KUKA KRL program: f1_Kuka_APT216T03S16.SRC

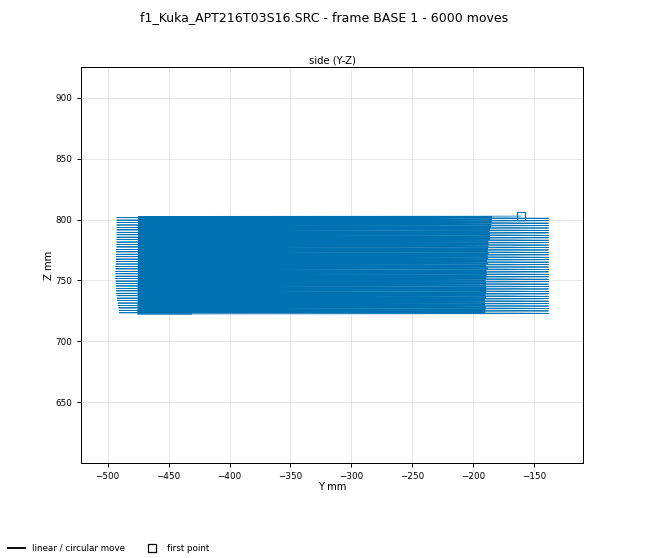
[picture p0: tool path of f1_Kuka_APT216T03S16.SRC in frame BASE 1, 6000 of 6001 moves have a stored position in this frame; points joined in program order, loops and branches not executed]
&ACCESS RVP
&REL 2
&PARAM TEMPLATE = C:\KRC\Roboter\Template\vorgabe
&PARAM EDITMASK = *
DEF f1_Kuka_APT216T03S16()


;FOLD INI;%{PE}%V3.2.0,%MKUKATPBASIS,%CINIT,%VCOMMON,%P
  ;FOLD BAS INI;%{E}%V3.2.0,%MKUKATPBASIS,%CINIT,%VINIT,%P
    GLOBAL INTERRUPT DECL 3 WHEN $STOPMESS==TRUE DO IR_STOPM ( )
    INTERRUPT ON 3
    BAS (#INITMOV,0 )
  ;ENDFOLD (BAS INI)
  ;FOLD USER INI;%{E}%V3.2.0,%MKUKATPUSER,%CINIT,%VINIT,%P
    ;Make your modifications here
  ;ENDFOLD (USER INI)
;ENDFOLD (INI)


;*** Make Null PTP Move
  PTP $pos_act

;*** Auto Load The Correct TOOL Data
  $tool=tool_data[3]

;*** Auto Load The Correct BASE Data
  $base=base_data[1]

  $ADVANCE = 5

;*** Restate Last Velocity
MMPM(30000.0)
SetRPM(6000)
LIN {X -0.024,Y -161.232,Z 802.830,A 0.000,B 0.000,C 90.000,E1 149.459} C_DIS
LIN {X 0.060,Y -163.319,Z 802.820,A 0.000,B 0.000,C 90.000,E1 147.661} C_DIS
LIN {X -0.068,Y -167.771,Z 802.801,A 0.000,B 0.000,C 90.000,E1 144.196} C_DIS
LIN {X 0.084,Y -171.586,Z 802.786,A 0.000,B 0.000,C 90.000,E1 141.537} C_DIS
LIN {X 0.015,Y -176.537,Z 802.767,A 0.000,B 0.000,C 90.000,E1 138.119} C_DIS
LIN {X 0.007,Y -180.836,Z 802.753,A 0.000,B 0.000,C 90.000,E1 135.567} C_DIS
LIN {X -0.008,Y -186.246,Z 802.734,A 0.000,B 0.000,C 90.000,E1 132.204} C_DIS
LIN {X -0.071,Y -190.882,Z 802.721,A 0.000,B 0.000,C 90.000,E1 129.725} C_DIS
LIN {X 0.062,Y -192.636,Z 802.715,A 0.000,B 0.000,C 90.000,E1 128.624} C_DIS
LIN {X 0.046,Y -293.294,Z 802.715,A 0.000,B 0.000,C 90.000,E1 128.624} C_DIS
LIN {X -0.102,Y -294.709,Z 802.714,A 0.000,B 0.000,C 90.000,E1 128.624} C_DIS
LIN {X -0.048,Y -299.870,Z 802.713,A 0.000,B 0.000,C 90.000,E1 128.338} C_DIS
LIN {X 0.009,Y -302.645,Z 802.711,A 0.000,B 0.000,C 90.000,E1 128.051} C_DIS
LIN {X -0.181,Y -306.338,Z 802.708,A 0.000,B 0.000,C 90.000,E1 127.523} C_DIS
LIN {X 0.019,Y -307.841,Z 802.706,A 0.000,B 0.000,C 90.000,E1 127.156} C_DIS
LIN {X 0.036,Y -309.022,Z 802.705,A 0.000,B 0.000,C 90.000,E1 126.824} C_DIS
LIN {X -0.142,Y -320.038,Z 802.685,A 0.000,B 0.000,C 90.000,E1 123.293} C_DIS
LIN {X -0.035,Y -330.415,Z 802.669,A 0.000,B 0.000,C 90.000,E1 120.413} C_DIS
LIN {X 0.057,Y -342.138,Z 802.653,A 0.000,B 0.000,C 90.000,E1 117.590} C_DIS
LIN {X 0.009,Y -355.318,Z 802.638,A 0.000,B 0.000,C 90.000,E1 114.847} C_DIS
LIN {X -0.042,Y -368.347,Z 802.625,A 0.000,B 0.000,C 90.000,E1 112.461} C_DIS
LIN {X -0.058,Y -382.712,Z 802.612,A 0.000,B 0.000,C 90.000,E1 110.120} C_DIS
LIN {X 0.023,Y -398.513,Z 802.599,A 0.000,B 0.000,C 90.000,E1 107.819} C_DIS
LIN {X -0.127,Y -415.866,Z 802.587,A 0.000,B 0.000,C 90.000,E1 105.607} C_DIS
LIN {X 0.032,Y -434.898,Z 802.575,A 0.000,B 0.000,C 90.000,E1 103.411} C_DIS
LIN {X 0.068,Y -454.991,Z 802.563,A 0.000,B 0.000,C 90.000,E1 101.366} C_DIS
LIN {X -0.083,Y -467.781,Z 802.557,A 0.000,B 0.000,C 90.000,E1 100.197} C_DIS
LIN {X -0.048,Y -469.816,Z 802.555,A 0.000,B 0.000,C 90.000,E1 99.962} C_DIS
LIN {X -0.200,Y -471.497,Z 802.554,A 0.000,B 0.000,C 90.000,E1 99.726} C_DIS
LIN {X 0.036,Y -472.760,Z 802.552,A 0.000,B 0.000,C 90.000,E1 99.443} C_DIS
LIN {X 0.218,Y -474.319,Z 802.550,A 0.000,B 0.000,C 90.000,E1 98.916} C_DIS
LIN {X -0.134,Y -474.830,Z 802.547,A 0.000,B 0.000,C 90.000,E1 98.454} C_DIS
LIN {X -0.007,Y -474.378,Z 802.544,A 0.000,B 0.000,C 90.000,E1 97.936} C_DIS
LIN {X 0.185,Y -472.896,Z 802.541,A 0.000,B 0.000,C 90.000,E1 97.409} C_DIS
LIN {X -0.015,Y -471.693,Z 802.540,A 0.000,B 0.000,C 90.000,E1 97.182} C_DIS
LIN {X 0.161,Y -454.007,Z 802.524,A 0.000,B 0.000,C 90.000,E1 94.359} C_DIS
LIN {X -0.210,Y -440.415,Z 802.511,A 0.000,B 0.000,C 90.000,E1 92.064} C_DIS
LIN {X -0.069,Y -431.096,Z 802.503,A 0.000,B 0.000,C 90.000,E1 90.458} C_DIS
LIN {X 0.016,Y -419.942,Z 802.492,A 0.000,B 0.000,C 90.000,E1 88.568} C_DIS
LIN {X -0.207,Y -410.228,Z 802.483,A 0.000,B 0.000,C 90.000,E1 86.963} C_DIS
LIN {X -0.090,Y -398.712,Z 802.472,A 0.000,B 0.000,C 90.000,E1 85.008} C_DIS
LIN {X -0.164,Y -385.665,Z 802.460,A 0.000,B 0.000,C 90.000,E1 82.761} C_DIS
LIN {X -0.060,Y -371.493,Z 802.445,A 0.000,B 0.000,C 90.000,E1 80.151} C_DIS
LIN {X 0.105,Y -356.306,Z 802.429,A 0.000,B 0.000,C 90.000,E1 77.173} C_DIS
LIN {X 0.123,Y -344.660,Z 802.415,A 0.000,B 0.000,C 90.000,E1 74.755} C_DIS
LIN {X 0.037,Y -333.108,Z 802.402,A 0.000,B 0.000,C 90.000,E1 72.308} C_DIS
LIN {X -0.175,Y -320.385,Z 802.386,A 0.000,B 0.000,C 90.000,E1 69.518} C_DIS
LIN {X -0.054,Y -306.773,Z 802.368,A 0.000,B 0.000,C 90.000,E1 66.282} C_DIS
LIN {X -0.094,Y -294.227,Z 802.350,A 0.000,B 0.000,C 90.000,E1 62.999} C_DIS
LIN {X 0.029,Y -283.577,Z 802.333,A 0.000,B 0.000,C 90.000,E1 59.950} C_DIS
LIN {X 0.171,Y -273.514,Z 802.316,A 0.000,B 0.000,C 90.000,E1 56.834} C_DIS
LIN {X 0.145,Y -265.985,Z 802.302,A 0.000,B 0.000,C 90.000,E1 54.402} C_DIS
LIN {X 0.011,Y -259.636,Z 802.291,A 0.000,B 0.000,C 90.000,E1 52.316} C_DIS
LIN {X -0.014,Y -251.225,Z 802.275,A 0.000,B 0.000,C 90.000,E1 49.461} C_DIS
LIN {X 0.018,Y -241.238,Z 802.255,A 0.000,B 0.000,C 90.000,E1 45.810} C_DIS
LIN {X 0.075,Y -232.062,Z 802.234,A 0.000,B 0.000,C 90.000,E1 42.081} C_DIS
LIN {X 0.021,Y -225.008,Z 802.217,A 0.000,B 0.000,C 90.000,E1 39.072} C_DIS
LIN {X 0.019,Y -216.511,Z 802.196,A 0.000,B 0.000,C 90.000,E1 35.231} C_DIS
LIN {X -0.068,Y -210.188,Z 802.178,A 0.000,B 0.000,C 90.000,E1 32.133} C_DIS
LIN {X 0.005,Y -204.534,Z 802.161,A 0.000,B 0.000,C 90.000,E1 28.949} C_DIS
LIN {X 0.099,Y -199.559,Z 802.143,A 0.000,B 0.000,C 90.000,E1 25.720} C_DIS
LIN {X -0.011,Y -195.325,Z 802.125,A 0.000,B 0.000,C 90.000,E1 22.514} C_DIS
LIN {X 0.021,Y -191.093,Z 802.102,A 0.000,B 0.000,C 90.000,E1 18.417} C_DIS
LIN {X -0.033,Y -187.480,Z 802.075,A 0.000,B 0.000,C 90.000,E1 13.480} C_DIS
LIN {X -0.067,Y -185.036,Z 802.038,A 0.000,B 0.000,C 90.000,E1 6.834} C_DIS
LIN {X 0.017,Y -186.593,Z 801.974,A 0.000,B 0.000,C 90.000,E1 355.355} C_DIS
LIN {X -0.039,Y -189.431,Z 801.947,A 0.000,B 0.000,C 90.000,E1 350.387} C_DIS
LIN {X 0.059,Y -193.534,Z 801.919,A 0.000,B 0.000,C 90.000,E1 345.408} C_DIS
LIN {X 0.027,Y -197.946,Z 801.896,A 0.000,B 0.000,C 90.000,E1 341.329} C_DIS
LIN {X 0.027,Y -203.325,Z 801.874,A 0.000,B 0.000,C 90.000,E1 337.283} C_DIS
LIN {X 0.047,Y -208.352,Z 801.856,A 0.000,B 0.000,C 90.000,E1 334.076} C_DIS
LIN {X -0.005,Y -214.072,Z 801.838,A 0.000,B 0.000,C 90.000,E1 330.923} C_DIS
LIN {X -0.088,Y -221.910,Z 801.817,A 0.000,B 0.000,C 90.000,E1 327.041} C_DIS
LIN {X 0.131,Y -228.708,Z 801.800,A 0.000,B 0.000,C 90.000,E1 323.909} C_DIS
LIN {X 0.035,Y -237.880,Z 801.779,A 0.000,B 0.000,C 90.000,E1 320.150} C_DIS
LIN {X -0.020,Y -246.975,Z 801.760,A 0.000,B 0.000,C 90.000,E1 316.824} C_DIS
LIN {X 0.009,Y -256.777,Z 801.742,A 0.000,B 0.000,C 90.000,E1 313.542} C_DIS
LIN {X -0.010,Y -267.270,Z 801.724,A 0.000,B 0.000,C 90.000,E1 310.334} C_DIS
LIN {X -0.144,Y -280.020,Z 801.705,A 0.000,B 0.000,C 90.000,E1 306.870} C_DIS
LIN {X -0.053,Y -291.202,Z 801.690,A 0.000,B 0.000,C 90.000,E1 304.119} C_DIS
LIN {X -0.149,Y -305.021,Z 801.673,A 0.000,B 0.000,C 90.000,E1 301.131} C_DIS
LIN {X -0.014,Y -316.931,Z 801.660,A 0.000,B 0.000,C 90.000,E1 298.821} C_DIS
LIN {X -0.144,Y -333.668,Z 801.644,A 0.000,B 0.000,C 90.000,E1 295.976} C_DIS
LIN {X 0.062,Y -349.615,Z 801.630,A 0.000,B 0.000,C 90.000,E1 293.462} C_DIS
LIN {X 0.090,Y -367.192,Z 801.617,A 0.000,B 0.000,C 90.000,E1 291.046} C_DIS
LIN {X 0.108,Y -391.664,Z 801.601,A 0.000,B 0.000,C 90.000,E1 288.127} C_DIS
LIN {X 0.031,Y -409.097,Z 801.590,A 0.000,B 0.000,C 90.000,E1 286.205} C_DIS
LIN {X 0.102,Y -421.589,Z 801.582,A 0.000,B 0.000,C 90.000,E1 284.828} C_DIS
LIN {X -0.046,Y -431.397,Z 801.576,A 0.000,B 0.000,C 90.000,E1 283.772} C_DIS
LIN {X 0.161,Y -443.375,Z 801.569,A 0.000,B 0.000,C 90.000,E1 282.411} C_DIS
LIN {X 0.111,Y -452.462,Z 801.563,A 0.000,B 0.000,C 90.000,E1 281.366} C_DIS
LIN {X -0.193,Y -460.841,Z 801.557,A 0.000,B 0.000,C 90.000,E1 280.366} C_DIS
LIN {X -0.037,Y -468.618,Z 801.552,A 0.000,B 0.000,C 90.000,E1 279.321} C_DIS
LIN {X -0.111,Y -474.039,Z 801.548,A 0.000,B 0.000,C 90.000,E1 278.568} C_DIS
LIN {X -0.134,Y -478.846,Z 801.543,A 0.000,B 0.000,C 90.000,E1 277.814} C_DIS
LIN {X -0.180,Y -482.999,Z 801.539,A 0.000,B 0.000,C 90.000,E1 277.068} C_DIS
LIN {X -0.125,Y -486.497,Z 801.535,A 0.000,B 0.000,C 90.000,E1 276.315} C_DIS
LIN {X -0.095,Y -489.290,Z 801.531,A 0.000,B 0.000,C 90.000,E1 275.568} C_DIS
LIN {X 0.114,Y -490.692,Z 801.528,A 0.000,B 0.000,C 90.000,E1 275.049} C_DIS
LIN {X -0.158,Y -491.677,Z 801.525,A 0.000,B 0.000,C 90.000,E1 274.588} C_DIS
LIN {X 0.032,Y -492.321,Z 801.523,A 0.000,B 0.000,C 90.000,E1 274.073} C_DIS
LIN {X -0.229,Y -492.497,Z 801.520,A 0.000,B 0.000,C 90.000,E1 273.612} C_DIS
LIN {X 0.001,Y -492.328,Z 801.517,A 0.000,B 0.000,C 90.000,E1 273.094} C_DIS
LIN {X 0.206,Y -491.749,Z 801.514,A 0.000,B 0.000,C 90.000,E1 272.579} C_DIS
LIN {X -0.079,Y -490.766,Z 801.512,A 0.000,B 0.000,C 90.000,E1 272.121} C_DIS
LIN {X 0.141,Y -489.390,Z 801.509,A 0.000,B 0.000,C 90.000,E1 271.604} C_DIS
LIN {X -0.150,Y -487.564,Z 801.506,A 0.000,B 0.000,C 90.000,E1 271.146} C_DIS
LIN {X 0.040,Y -485.253,Z 801.504,A 0.000,B 0.000,C 90.000,E1 270.630} C_DIS
LIN {X 0.212,Y -482.387,Z 801.501,A 0.000,B 0.000,C 90.000,E1 270.115} C_DIS
LIN {X -0.110,Y -478.964,Z 801.498,A 0.000,B 0.000,C 90.000,E1 269.656} C_DIS
LIN {X 0.029,Y -474.681,Z 801.495,A 0.000,B 0.000,C 90.000,E1 269.141} C_DIS
LIN {X 0.143,Y -469.391,Z 801.492,A 0.000,B 0.000,C 90.000,E1 268.625} C_DIS
LIN {X 0.125,Y -466.571,Z 801.491,A 0.000,B 0.000,C 90.000,E1 268.396} C_DIS
LIN {X -0.091,Y -460.311,Z 801.489,A 0.000,B 0.000,C 90.000,E1 267.993} C_DIS
LIN {X 0.156,Y -456.765,Z 801.488,A 0.000,B 0.000,C 90.000,E1 267.764} C_DIS
LIN {X -0.162,Y -449.428,Z 801.486,A 0.000,B 0.000,C 90.000,E1 267.478} C_DIS
LIN {X 0.099,Y -441.906,Z 801.484,A 0.000,B 0.000,C 90.000,E1 267.192} C_DIS
LIN {X -0.084,Y -433.510,Z 801.483,A 0.000,B 0.000,C 90.000,E1 267.020} C_DIS
LIN {X 0.009,Y -425.926,Z 801.483,A 0.000,B 0.000,C 90.000,E1 266.906} C_DIS
LIN {X 0.122,Y -418.652,Z 801.483,A 0.000,B 0.000,C 90.000,E1 266.849} C_DIS
LIN {X 0.039,Y -180.978,Z 801.483,A 0.000,B 0.000,C 90.000,E1 266.846} C_DIS
LIN {X 0.015,Y -180.886,Z 801.473,A 0.000,B 0.000,C 90.000,E1 265.122} C_DIS
LIN {X 0.074,Y -179.008,Z 801.445,A 0.000,B 0.000,C 90.000,E1 260.038} C_DIS
LIN {X -0.008,Y -178.618,Z 801.440,A 0.000,B 0.000,C 90.000,E1 259.218} C_DIS
LIN {X 0.060,Y -175.670,Z 801.412,A 0.000,B 0.000,C 90.000,E1 254.102} C_DIS
LIN {X 0.065,Y -172.386,Z 801.388,A 0.000,B 0.000,C 90.000,E1 249.826} C_DIS
LIN {X 0.079,Y -171.189,Z 801.378,A 0.000,B 0.000,C 90.000,E1 248.103} C_DIS
LIN {X -0.029,Y -167.480,Z 801.354,A 0.000,B 0.000,C 90.000,E1 243.819} C_DIS
LIN {X -0.021,Y -166.876,Z 801.350,A 0.000,B 0.000,C 90.000,E1 242.948} C_DIS
LIN {X -0.028,Y -162.181,Z 801.321,A 0.000,B 0.000,C 90.000,E1 237.709} C_DIS
LIN {X 0.029,Y -160.748,Z 801.311,A 0.000,B 0.000,C 90.000,E1 235.928} C_DIS
LIN {X 0.007,Y -157.548,Z 801.291,A 0.000,B 0.000,C 90.000,E1 232.396} C_DIS
LIN {X -0.054,Y -155.576,Z 801.276,A 0.000,B 0.000,C 90.000,E1 229.747} C_DIS
LIN {X -0.002,Y -151.861,Z 801.251,A 0.000,B 0.000,C 90.000,E1 225.243} C_DIS
LIN {X 0.012,Y -150.084,Z 801.236,A 0.000,B 0.000,C 90.000,E1 222.528} C_DIS
LIN {X 0.046,Y -146.887,Z 801.211,A 0.000,B 0.000,C 90.000,E1 217.971} C_DIS
LIN {X 0.034,Y -145.473,Z 801.196,A 0.000,B 0.000,C 90.000,E1 215.231} C_DIS
LIN {X -0.049,Y -142.884,Z 801.170,A 0.000,B 0.000,C 90.000,E1 210.669} C_DIS
LIN {X 0.008,Y -141.503,Z 801.150,A 0.000,B 0.000,C 90.000,E1 206.950} C_DIS
LIN {X 0.056,Y -139.389,Z 801.114,A 0.000,B 0.000,C 90.000,E1 200.429} C_DIS
LIN {X -0.024,Y -139.096,Z 801.103,A 0.000,B 0.000,C 90.000,E1 198.598} C_DIS
LIN {X -0.031,Y -138.354,Z 801.057,A 0.000,B 0.000,C 90.000,E1 190.197} C_DIS
LIN {X -0.039,Y -139.516,Z 801.005,A 0.000,B 0.000,C 90.000,E1 180.859} C_DIS
LIN {X 0.042,Y -141.170,Z 800.974,A 0.000,B 0.000,C 90.000,E1 175.241} C_DIS
LIN {X 0.013,Y -142.550,Z 800.958,A 0.000,B 0.000,C 90.000,E1 172.470} C_DIS
LIN {X -0.061,Y -144.825,Z 800.933,A 0.000,B 0.000,C 90.000,E1 167.881} C_DIS
LIN {X 0.067,Y -147.448,Z 800.912,A 0.000,B 0.000,C 90.000,E1 164.157} C_DIS
LIN {X -0.046,Y -150.029,Z 800.892,A 0.000,B 0.000,C 90.000,E1 160.550} C_DIS
LIN {X -0.040,Y -153.365,Z 800.872,A 0.000,B 0.000,C 90.000,E1 156.922} C_DIS
LIN {X 0.008,Y -155.899,Z 800.857,A 0.000,B 0.000,C 90.000,E1 154.204} C_DIS
LIN {X -0.094,Y -159.759,Z 800.837,A 0.000,B 0.000,C 90.000,E1 150.667} C_DIS
LIN {X -0.028,Y -161.999,Z 800.827,A 0.000,B 0.000,C 90.000,E1 148.869} C_DIS
LIN {X -0.009,Y -166.192,Z 800.807,A 0.000,B 0.000,C 90.000,E1 145.341} C_DIS
LIN {X 0.088,Y -171.207,Z 800.788,A 0.000,B 0.000,C 90.000,E1 141.823} C_DIS
LIN {X 0.013,Y -176.091,Z 800.769,A 0.000,B 0.000,C 90.000,E1 138.405} C_DIS
LIN {X 0.005,Y -180.352,Z 800.755,A 0.000,B 0.000,C 90.000,E1 135.850} C_DIS
LIN {X 0.108,Y -185.762,Z 800.736,A 0.000,B 0.000,C 90.000,E1 132.447} C_DIS
LIN {X -0.105,Y -190.374,Z 800.722,A 0.000,B 0.000,C 90.000,E1 130.011} C_DIS
LIN {X -0.053,Y -192.619,Z 800.715,A 0.000,B 0.000,C 90.000,E1 128.669} C_DIS
LIN {X -0.111,Y -292.511,Z 800.715,A 0.000,B 0.000,C 90.000,E1 128.669} C_DIS
LIN {X 0.124,Y -297.634,Z 800.714,A 0.000,B 0.000,C 90.000,E1 128.463} C_DIS
LIN {X -0.057,Y -299.936,Z 800.713,A 0.000,B 0.000,C 90.000,E1 128.338} C_DIS
LIN {X 0.094,Y -303.787,Z 800.711,A 0.000,B 0.000,C 90.000,E1 127.890} C_DIS
LIN {X 0.015,Y -305.707,Z 800.709,A 0.000,B 0.000,C 90.000,E1 127.604} C_DIS
LIN {X -0.067,Y -307.217,Z 800.707,A 0.000,B 0.000,C 90.000,E1 127.317} C_DIS
LIN {X 0.145,Y -308.517,Z 800.705,A 0.000,B 0.000,C 90.000,E1 126.950} C_DIS
LIN {X 0.026,Y -320.615,Z 800.684,A 0.000,B 0.000,C 90.000,E1 123.086} C_DIS
LIN {X -0.131,Y -331.071,Z 800.668,A 0.000,B 0.000,C 90.000,E1 120.256} C_DIS
LIN {X -0.037,Y -342.880,Z 800.652,A 0.000,B 0.000,C 90.000,E1 117.436} C_DIS
LIN {X -0.081,Y -356.152,Z 800.637,A 0.000,B 0.000,C 90.000,E1 114.695} C_DIS
LIN {X 0.070,Y -369.271,Z 800.624,A 0.000,B 0.000,C 90.000,E1 112.280} C_DIS
LIN {X 0.085,Y -383.730,Z 800.611,A 0.000,B 0.000,C 90.000,E1 109.939} C_DIS
LIN {X 0.199,Y -399.636,Z 800.598,A 0.000,B 0.000,C 90.000,E1 107.638} C_DIS
LIN {X 0.082,Y -417.100,Z 800.586,A 0.000,B 0.000,C 90.000,E1 105.426} C_DIS
LIN {X -0.234,Y -436.237,Z 800.574,A 0.000,B 0.000,C 90.000,E1 103.300} C_DIS
LIN {X -0.019,Y -456.369,Z 800.562,A 0.000,B 0.000,C 90.000,E1 101.243} C_DIS
LIN {X -0.165,Y -466.643,Z 800.557,A 0.000,B 0.000,C 90.000,E1 100.310} C_DIS
LIN {X -0.121,Y -468.956,Z 800.556,A 0.000,B 0.000,C 90.000,E1 100.074} C_DIS
LIN {X -0.157,Y -470.704,Z 800.555,A 0.000,B 0.000,C 90.000,E1 99.849} C_DIS
LIN {X 0.160,Y -472.169,Z 800.553,A 0.000,B 0.000,C 90.000,E1 99.557} C_DIS
LIN {X 0.011,Y -473.263,Z 800.552,A 0.000,B 0.000,C 90.000,E1 99.321} C_DIS
LIN {X 0.123,Y -474.554,Z 800.549,A 0.000,B 0.000,C 90.000,E1 98.803} C_DIS
LIN {X -0.227,Y -474.834,Z 800.546,A 0.000,B 0.000,C 90.000,E1 98.341} C_DIS
LIN {X -0.032,Y -474.148,Z 800.543,A 0.000,B 0.000,C 90.000,E1 97.814} C_DIS
LIN {X 0.097,Y -472.391,Z 800.541,A 0.000,B 0.000,C 90.000,E1 97.296} C_DIS
LIN {X -0.103,Y -471.010,Z 800.539,A 0.000,B 0.000,C 90.000,E1 97.068} C_DIS
LIN {X 0.066,Y -456.340,Z 800.526,A 0.000,B 0.000,C 90.000,E1 94.759} C_DIS
LIN {X 0.190,Y -442.717,Z 800.513,A 0.000,B 0.000,C 90.000,E1 92.407} C_DIS
LIN {X 0.204,Y -435.039,Z 800.506,A 0.000,B 0.000,C 90.000,E1 91.088} C_DIS
LIN {X -0.194,Y -425.570,Z 800.497,A 0.000,B 0.000,C 90.000,E1 89.542} C_DIS
LIN {X 0.106,Y -415.962,Z 800.488,A 0.000,B 0.000,C 90.000,E1 87.879} C_DIS
LIN {X -0.183,Y -406.168,Z 800.479,A 0.000,B 0.000,C 90.000,E1 86.274} C_DIS
LIN {X -0.146,Y -394.667,Z 800.468,A 0.000,B 0.000,C 90.000,E1 84.318} C_DIS
LIN {X 0.091,Y -380.170,Z 800.454,A 0.000,B 0.000,C 90.000,E1 81.724} C_DIS
LIN {X 0.107,Y -369.241,Z 800.443,A 0.000,B 0.000,C 90.000,E1 79.690} C_DIS
LIN {X -0.109,Y -355.684,Z 800.428,A 0.000,B 0.000,C 90.000,E1 77.061} C_DIS
LIN {X -0.015,Y -344.035,Z 800.415,A 0.000,B 0.000,C 90.000,E1 74.629} C_DIS
LIN {X -0.106,Y -332.517,Z 800.401,A 0.000,B 0.000,C 90.000,E1 72.181} C_DIS
LIN {X -0.023,Y -319.833,Z 800.385,A 0.000,B 0.000,C 90.000,E1 69.337} C_DIS
LIN {X -0.020,Y -305.018,Z 800.365,A 0.000,B 0.000,C 90.000,E1 65.793} C_DIS
LIN {X 0.006,Y -292.639,Z 800.347,A 0.000,B 0.000,C 90.000,E1 62.487} C_DIS
LIN {X 0.004,Y -283.251,Z 800.332,A 0.000,B 0.000,C 90.000,E1 59.793} C_DIS
LIN {X 0.057,Y -274.379,Z 800.317,A 0.000,B 0.000,C 90.000,E1 57.041} C_DIS
LIN {X -0.018,Y -265.800,Z 800.302,A 0.000,B 0.000,C 90.000,E1 54.276} C_DIS
LIN {X 0.050,Y -259.485,Z 800.290,A 0.000,B 0.000,C 90.000,E1 52.145} C_DIS
LIN {X -0.022,Y -251.109,Z 800.274,A 0.000,B 0.000,C 90.000,E1 49.299} C_DIS
LIN {X 0.010,Y -241.186,Z 800.254,A 0.000,B 0.000,C 90.000,E1 45.648} C_DIS
LIN {X 0.064,Y -232.032,Z 800.233,A 0.000,B 0.000,C 90.000,E1 41.919} C_DIS
LIN {X 0.007,Y -224.973,Z 800.216,A 0.000,B 0.000,C 90.000,E1 38.910} C_DIS
LIN {X -0.125,Y -216.490,Z 800.195,A 0.000,B 0.000,C 90.000,E1 35.105} C_DIS
LIN {X 0.084,Y -210.177,Z 800.177,A 0.000,B 0.000,C 90.000,E1 31.926} C_DIS
LIN {X -0.127,Y -204.556,Z 800.160,A 0.000,B 0.000,C 90.000,E1 28.821} C_DIS
LIN {X -0.030,Y -199.636,Z 800.142,A 0.000,B 0.000,C 90.000,E1 25.591} C_DIS
LIN {X 0.045,Y -195.431,Z 800.124,A 0.000,B 0.000,C 90.000,E1 22.333} C_DIS
LIN {X 0.081,Y -191.215,Z 800.101,A 0.000,B 0.000,C 90.000,E1 18.236} C_DIS
LIN {X 0.029,Y -187.650,Z 800.074,A 0.000,B 0.000,C 90.000,E1 13.300} C_DIS
LIN {X -0.028,Y -185.241,Z 800.037,A 0.000,B 0.000,C 90.000,E1 6.663} C_DIS
LIN {X 0.023,Y -186.790,Z 799.974,A 0.000,B 0.000,C 90.000,E1 355.355} C_DIS
LIN {X -0.051,Y -190.199,Z 799.942,A 0.000,B 0.000,C 90.000,E1 349.567} C_DIS
LIN {X 0.079,Y -193.692,Z 799.919,A 0.000,B 0.000,C 90.000,E1 345.408} C_DIS
LIN {X 0.053,Y -198.100,Z 799.896,A 0.000,B 0.000,C 90.000,E1 341.329} C_DIS
LIN {X -0.020,Y -203.489,Z 799.874,A 0.000,B 0.000,C 90.000,E1 337.305} C_DIS
LIN {X -0.009,Y -208.529,Z 799.856,A 0.000,B 0.000,C 90.000,E1 334.101} C_DIS
LIN {X 0.036,Y -214.254,Z 799.839,A 0.000,B 0.000,C 90.000,E1 330.923} C_DIS
LIN {X -0.039,Y -222.077,Z 799.817,A 0.000,B 0.000,C 90.000,E1 327.041} C_DIS
LIN {X -0.133,Y -228.854,Z 799.800,A 0.000,B 0.000,C 90.000,E1 323.989} C_DIS
LIN {X -0.085,Y -238.010,Z 799.779,A 0.000,B 0.000,C 90.000,E1 320.194} C_DIS
LIN {X 0.047,Y -247.073,Z 799.760,A 0.000,B 0.000,C 90.000,E1 316.824} C_DIS
LIN {X 0.082,Y -256.834,Z 799.742,A 0.000,B 0.000,C 90.000,E1 313.542} C_DIS
LIN {X -0.072,Y -268.523,Z 799.722,A 0.000,B 0.000,C 90.000,E1 310.011} C_DIS
LIN {X 0.045,Y -281.342,Z 799.703,A 0.000,B 0.000,C 90.000,E1 306.503} C_DIS
LIN {X 0.148,Y -295.599,Z 799.684,A 0.000,B 0.000,C 90.000,E1 303.086} C_DIS
LIN {X -0.005,Y -308.256,Z 799.669,A 0.000,B 0.000,C 90.000,E1 300.463} C_DIS
LIN {X 0.055,Y -320.454,Z 799.657,A 0.000,B 0.000,C 90.000,E1 298.180} C_DIS
LIN {X 0.033,Y -337.394,Z 799.641,A 0.000,B 0.000,C 90.000,E1 295.335} C_DIS
LIN {X -0.144,Y -351.561,Z 799.629,A 0.000,B 0.000,C 90.000,E1 293.206} C_DIS
LIN {X -0.158,Y -366.987,Z 799.617,A 0.000,B 0.000,C 90.000,E1 291.099} C_DIS
LIN {X -0.171,Y -391.384,Z 799.601,A 0.000,B 0.000,C 90.000,E1 288.181} C_DIS
LIN {X -0.062,Y -408.999,Z 799.590,A 0.000,B 0.000,C 90.000,E1 286.205} C_DIS
LIN {X 0.050,Y -421.432,Z 799.582,A 0.000,B 0.000,C 90.000,E1 284.828} C_DIS
LIN {X 0.006,Y -433.704,Z 799.575,A 0.000,B 0.000,C 90.000,E1 283.480} C_DIS
LIN {X 0.244,Y -445.594,Z 799.568,A 0.000,B 0.000,C 90.000,E1 282.119} C_DIS
LIN {X -0.222,Y -454.526,Z 799.562,A 0.000,B 0.000,C 90.000,E1 281.130} C_DIS
LIN {X -0.058,Y -462.740,Z 799.556,A 0.000,B 0.000,C 90.000,E1 280.074} C_DIS
LIN {X 0.123,Y -470.367,Z 799.550,A 0.000,B 0.000,C 90.000,E1 279.029} C_DIS
LIN {X 0.071,Y -475.598,Z 799.546,A 0.000,B 0.000,C 90.000,E1 278.276} C_DIS
LIN {X -0.006,Y -480.214,Z 799.542,A 0.000,B 0.000,C 90.000,E1 277.530} C_DIS
LIN {X 0.027,Y -484.170,Z 799.538,A 0.000,B 0.000,C 90.000,E1 276.777} C_DIS
LIN {X 0.037,Y -487.462,Z 799.534,A 0.000,B 0.000,C 90.000,E1 276.030} C_DIS
LIN {X -0.246,Y -489.184,Z 799.531,A 0.000,B 0.000,C 90.000,E1 275.568} C_DIS
LIN {X -0.038,Y -490.610,Z 799.528,A 0.000,B 0.000,C 90.000,E1 275.049} C_DIS
LIN {X 0.179,Y -491.646,Z 799.525,A 0.000,B 0.000,C 90.000,E1 274.531} C_DIS
LIN {X -0.122,Y -492.287,Z 799.523,A 0.000,B 0.000,C 90.000,E1 274.073} C_DIS
LIN {X 0.109,Y -492.502,Z 799.520,A 0.000,B 0.000,C 90.000,E1 273.555} C_DIS
LIN {X -0.153,Y -492.343,Z 799.517,A 0.000,B 0.000,C 90.000,E1 273.094} C_DIS
LIN {X 0.052,Y -491.743,Z 799.514,A 0.000,B 0.000,C 90.000,E1 272.579} C_DIS
LIN {X -0.232,Y -490.788,Z 799.512,A 0.000,B 0.000,C 90.000,E1 272.121} C_DIS
LIN {X -0.012,Y -489.386,Z 799.509,A 0.000,B 0.000,C 90.000,E1 271.604} C_DIS
LIN {X 0.185,Y -487.561,Z 799.506,A 0.000,B 0.000,C 90.000,E1 271.088} C_DIS
LIN {X -0.111,Y -485.243,Z 799.503,A 0.000,B 0.000,C 90.000,E1 270.630} C_DIS
LIN {X 0.062,Y -482.413,Z 799.501,A 0.000,B 0.000,C 90.000,E1 270.115} C_DIS
LIN {X 0.219,Y -478.949,Z 799.498,A 0.000,B 0.000,C 90.000,E1 269.599} C_DIS
LIN {X -0.120,Y -474.674,Z 799.495,A 0.000,B 0.000,C 90.000,E1 269.141} C_DIS
LIN {X -0.004,Y -469.439,Z 799.492,A 0.000,B 0.000,C 90.000,E1 268.625} C_DIS
LIN {X -0.058,Y -463.323,Z 799.490,A 0.000,B 0.000,C 90.000,E1 268.165} C_DIS
LIN {X 0.176,Y -460.210,Z 799.489,A 0.000,B 0.000,C 90.000,E1 267.936} C_DIS
LIN {X -0.052,Y -456.648,Z 799.488,A 0.000,B 0.000,C 90.000,E1 267.764} C_DIS
LIN {X 0.073,Y -449.208,Z 799.486,A 0.000,B 0.000,C 90.000,E1 267.421} C_DIS
LIN {X -0.014,Y -445.834,Z 799.485,A 0.000,B 0.000,C 90.000,E1 267.306} C_DIS
LIN {X 0.058,Y -438.104,Z 799.484,A 0.000,B 0.000,C 90.000,E1 267.078} C_DIS
LIN {X -0.222,Y -433.591,Z 799.483,A 0.000,B 0.000,C 90.000,E1 267.020} C_DIS
LIN {X -0.104,Y -426.050,Z 799.483,A 0.000,B 0.000,C 90.000,E1 266.906} C_DIS
LIN {X 0.040,Y -419.630,Z 799.482,A 0.000,B 0.000,C 90.000,E1 266.846} C_DIS
LIN {X -0.007,Y -180.977,Z 799.482,A 0.000,B 0.000,C 90.000,E1 266.846} C_DIS
LIN {X -0.039,Y -180.883,Z 799.473,A 0.000,B 0.000,C 90.000,E1 265.122} C_DIS
LIN {X 0.020,Y -179.003,Z 799.445,A 0.000,B 0.000,C 90.000,E1 260.038} C_DIS
LIN {X -0.061,Y -178.605,Z 799.440,A 0.000,B 0.000,C 90.000,E1 259.218} C_DIS
LIN {X 0.007,Y -175.658,Z 799.412,A 0.000,B 0.000,C 90.000,E1 254.102} C_DIS
LIN {X 0.013,Y -172.376,Z 799.388,A 0.000,B 0.000,C 90.000,E1 249.826} C_DIS
LIN {X 0.027,Y -171.171,Z 799.378,A 0.000,B 0.000,C 90.000,E1 248.103} C_DIS
LIN {X 0.071,Y -167.467,Z 799.354,A 0.000,B 0.000,C 90.000,E1 243.768} C_DIS
LIN {X 0.004,Y -166.864,Z 799.350,A 0.000,B 0.000,C 90.000,E1 242.922} C_DIS
LIN {X 0.058,Y -162.168,Z 799.320,A 0.000,B 0.000,C 90.000,E1 237.661} C_DIS
LIN {X -0.021,Y -160.730,Z 799.311,A 0.000,B 0.000,C 90.000,E1 235.928} C_DIS
LIN {X -0.042,Y -157.533,Z 799.291,A 0.000,B 0.000,C 90.000,E1 232.396} C_DIS
LIN {X 0.015,Y -155.559,Z 799.276,A 0.000,B 0.000,C 90.000,E1 229.703} C_DIS
LIN {X -0.051,Y -151.849,Z 799.251,A 0.000,B 0.000,C 90.000,E1 225.243} C_DIS
LIN {X -0.036,Y -150.068,Z 799.236,A 0.000,B 0.000,C 90.000,E1 222.528} C_DIS
LIN {X -0.002,Y -146.876,Z 799.211,A 0.000,B 0.000,C 90.000,E1 217.971} C_DIS
LIN {X -0.013,Y -145.462,Z 799.196,A 0.000,B 0.000,C 90.000,E1 215.231} C_DIS
LIN {X 0.028,Y -142.877,Z 799.170,A 0.000,B 0.000,C 90.000,E1 210.620} C_DIS
LIN {X 0.026,Y -141.494,Z 799.150,A 0.000,B 0.000,C 90.000,E1 206.924} C_DIS
LIN {X 0.010,Y -139.386,Z 799.114,A 0.000,B 0.000,C 90.000,E1 200.429} C_DIS
LIN {X -0.001,Y -138.843,Z 799.098,A 0.000,B 0.000,C 90.000,E1 197.638} C_DIS
LIN {X 0.059,Y -138.354,Z 799.056,A 0.000,B 0.000,C 90.000,E1 190.141} C_DIS
LIN {X 0.055,Y -139.519,Z 799.005,A 0.000,B 0.000,C 90.000,E1 180.802} C_DIS
LIN {X -0.004,Y -141.178,Z 798.974,A 0.000,B 0.000,C 90.000,E1 175.241} C_DIS
LIN {X -0.033,Y -142.557,Z 798.958,A 0.000,B 0.000,C 90.000,E1 172.470} C_DIS
LIN {X 0.033,Y -144.837,Z 798.932,A 0.000,B 0.000,C 90.000,E1 167.825} C_DIS
LIN {X 0.020,Y -147.460,Z 798.912,A 0.000,B 0.000,C 90.000,E1 164.157} C_DIS
LIN {X 0.047,Y -150.044,Z 798.892,A 0.000,B 0.000,C 90.000,E1 160.496} C_DIS
LIN {X 0.052,Y -153.385,Z 798.872,A 0.000,B 0.000,C 90.000,E1 156.869} C_DIS
LIN {X -0.041,Y -155.916,Z 798.857,A 0.000,B 0.000,C 90.000,E1 154.204} C_DIS
LIN {X 0.073,Y -159.780,Z 798.837,A 0.000,B 0.000,C 90.000,E1 150.589} C_DIS
LIN {X -0.079,Y -162.020,Z 798.827,A 0.000,B 0.000,C 90.000,E1 148.869} C_DIS
LIN {X 0.034,Y -166.215,Z 798.807,A 0.000,B 0.000,C 90.000,E1 145.308} C_DIS
LIN {X 0.036,Y -171.231,Z 798.788,A 0.000,B 0.000,C 90.000,E1 141.823} C_DIS
LIN {X -0.040,Y -176.118,Z 798.769,A 0.000,B 0.000,C 90.000,E1 138.405} C_DIS
LIN {X 0.076,Y -180.383,Z 798.755,A 0.000,B 0.000,C 90.000,E1 135.810} C_DIS
LIN {X 0.053,Y -185.790,Z 798.736,A 0.000,B 0.000,C 90.000,E1 132.447} C_DIS
LIN {X -0.014,Y -190.408,Z 798.722,A 0.000,B 0.000,C 90.000,E1 129.967} C_DIS
LIN {X -0.029,Y -192.606,Z 798.715,A 0.000,B 0.000,C 90.000,E1 128.669} C_DIS
LIN {X -0.073,Y -292.432,Z 798.715,A 0.000,B 0.000,C 90.000,E1 128.669} C_DIS
LIN {X 0.035,Y -294.111,Z 798.715,A 0.000,B 0.000,C 90.000,E1 128.624} C_DIS
LIN {X 0.039,Y -297.991,Z 798.714,A 0.000,B 0.000,C 90.000,E1 128.463} C_DIS
LIN {X 0.042,Y -300.175,Z 798.713,A 0.000,B 0.000,C 90.000,E1 128.302} C_DIS
LIN {X -0.101,Y -304.057,Z 798.710,A 0.000,B 0.000,C 90.000,E1 127.890} C_DIS
LIN {X -0.043,Y -305.955,Z 798.709,A 0.000,B 0.000,C 90.000,E1 127.569} C_DIS
LIN {X 0.070,Y -307.446,Z 798.707,A 0.000,B 0.000,C 90.000,E1 127.237} C_DIS
LIN {X -0.149,Y -308.687,Z 798.705,A 0.000,B 0.000,C 90.000,E1 126.950} C_DIS
LIN {X -0.082,Y -319.693,Z 798.685,A 0.000,B 0.000,C 90.000,E1 123.372} C_DIS
LIN {X 0.193,Y -330.026,Z 798.669,A 0.000,B 0.000,C 90.000,E1 120.463} C_DIS
LIN {X -0.033,Y -341.707,Z 798.654,A 0.000,B 0.000,C 90.000,E1 117.692} C_DIS
LIN {X -0.107,Y -354.836,Z 798.639,A 0.000,B 0.000,C 90.000,E1 114.951} C_DIS
LIN {X 0.152,Y -367.821,Z 798.625,A 0.000,B 0.000,C 90.000,E1 112.514} C_DIS
LIN {X 0.125,Y -382.135,Z 798.612,A 0.000,B 0.000,C 90.000,E1 110.174} C_DIS
LIN {X 0.195,Y -397.884,Z 798.599,A 0.000,B 0.000,C 90.000,E1 107.873} C_DIS
LIN {X 0.031,Y -415.180,Z 798.587,A 0.000,B 0.000,C 90.000,E1 105.662} C_DIS
LIN {X 0.084,Y -434.139,Z 798.575,A 0.000,B 0.000,C 90.000,E1 103.480} C_DIS
LIN {X 0.172,Y -454.209,Z 798.564,A 0.000,B 0.000,C 90.000,E1 101.422} C_DIS
LIN {X -0.027,Y -467.052,Z 798.557,A 0.000,B 0.000,C 90.000,E1 100.254} C_DIS
LIN {X 0.021,Y -469.268,Z 798.556,A 0.000,B 0.000,C 90.000,E1 100.018} C_DIS
LIN {X -0.011,Y -470.944,Z 798.554,A 0.000,B 0.000,C 90.000,E1 99.792} C_DIS
LIN {X -0.158,Y -472.353,Z 798.553,A 0.000,B 0.000,C 90.000,E1 99.557} C_DIS
LIN {X 0.161,Y -473.401,Z 798.552,A 0.000,B 0.000,C 90.000,E1 99.265} C_DIS
LIN {X -0.195,Y -474.620,Z 798.549,A 0.000,B 0.000,C 90.000,E1 98.803} C_DIS
LIN {X -0.005,Y -474.834,Z 798.546,A 0.000,B 0.000,C 90.000,E1 98.276} C_DIS
LIN {X 0.122,Y -474.081,Z 798.543,A 0.000,B 0.000,C 90.000,E1 97.757} C_DIS
LIN {X -0.218,Y -472.241,Z 798.540,A 0.000,B 0.000,C 90.000,E1 97.296} C_DIS
LIN {X 0.108,Y -470.806,Z 798.539,A 0.000,B 0.000,C 90.000,E1 97.004} C_DIS
LIN {X 0.212,Y -456.127,Z 798.526,A 0.000,B 0.000,C 90.000,E1 94.702} C_DIS
LIN {X -0.115,Y -442.502,Z 798.513,A 0.000,B 0.000,C 90.000,E1 92.407} C_DIS
LIN {X -0.098,Y -434.835,Z 798.506,A 0.000,B 0.000,C 90.000,E1 91.088} C_DIS
LIN {X -0.068,Y -425.359,Z 798.497,A 0.000,B 0.000,C 90.000,E1 89.484} C_DIS
LIN {X -0.191,Y -415.745,Z 798.488,A 0.000,B 0.000,C 90.000,E1 87.879} C_DIS
LIN {X -0.070,Y -405.966,Z 798.479,A 0.000,B 0.000,C 90.000,E1 86.216} C_DIS
LIN {X -0.043,Y -394.478,Z 798.468,A 0.000,B 0.000,C 90.000,E1 84.261} C_DIS
LIN {X -0.193,Y -380.023,Z 798.454,A 0.000,B 0.000,C 90.000,E1 81.724} C_DIS
LIN {X -0.175,Y -367.549,Z 798.441,A 0.000,B 0.000,C 90.000,E1 79.398} C_DIS
LIN {X -0.003,Y -354.081,Z 798.426,A 0.000,B 0.000,C 90.000,E1 76.700} C_DIS
LIN {X -0.036,Y -342.476,Z 798.413,A 0.000,B 0.000,C 90.000,E1 74.283} C_DIS
LIN {X -0.072,Y -330.992,Z 798.399,A 0.000,B 0.000,C 90.000,E1 71.819} C_DIS
LIN {X 0.137,Y -319.751,Z 798.385,A 0.000,B 0.000,C 90.000,E1 69.263} C_DIS
LIN {X 0.016,Y -304.998,Z 798.365,A 0.000,B 0.000,C 90.000,E1 65.741} C_DIS
LIN {X 0.032,Y -292.659,Z 798.347,A 0.000,B 0.000,C 90.000,E1 62.436} C_DIS
LIN {X -0.009,Y -282.184,Z 798.330,A 0.000,B 0.000,C 90.000,E1 59.410} C_DIS
LIN {X 0.072,Y -274.517,Z 798.317,A 0.000,B 0.000,C 90.000,E1 56.993} C_DIS
LIN {X 0.147,Y -265.977,Z 798.301,A 0.000,B 0.000,C 90.000,E1 54.196} C_DIS
LIN {X 0.011,Y -259.683,Z 798.289,A 0.000,B 0.000,C 90.000,E1 52.110} C_DIS
LIN {X -0.017,Y -251.353,Z 798.274,A 0.000,B 0.000,C 90.000,E1 49.256} C_DIS
LIN {X 0.012,Y -241.454,Z 798.253,A 0.000,B 0.000,C 90.000,E1 45.607} C_DIS
LIN {X -0.092,Y -232.294,Z 798.233,A 0.000,B 0.000,C 90.000,E1 41.919} C_DIS
LIN {X 0.004,Y -225.233,Z 798.216,A 0.000,B 0.000,C 90.000,E1 38.874} C_DIS
LIN {X 0.044,Y -216.742,Z 798.195,A 0.000,B 0.000,C 90.000,E1 35.025} C_DIS
LIN {X -0.038,Y -210.433,Z 798.177,A 0.000,B 0.000,C 90.000,E1 31.926} C_DIS
LIN {X 0.038,Y -204.806,Z 798.160,A 0.000,B 0.000,C 90.000,E1 28.743} C_DIS
LIN {X 0.047,Y -199.906,Z 798.142,A 0.000,B 0.000,C 90.000,E1 25.540} C_DIS
LIN {X -0.102,Y -194.758,Z 798.119,A 0.000,B 0.000,C 90.000,E1 21.535} C_DIS
LIN {X 0.037,Y -190.760,Z 798.097,A 0.000,B 0.000,C 90.000,E1 17.402} C_DIS
LIN {X -0.072,Y -187.457,Z 798.069,A 0.000,B 0.000,C 90.000,E1 12.479} C_DIS
LIN {X -0.081,Y -185.256,Z 798.028,A 0.000,B 0.000,C 90.000,E1 4.992} C_DIS
LIN {X 0.029,Y -186.982,Z 797.974,A 0.000,B 0.000,C 90.000,E1 355.355} C_DIS
LIN {X -0.036,Y -190.368,Z 797.942,A 0.000,B 0.000,C 90.000,E1 349.567} C_DIS
LIN {X -0.089,Y -193.845,Z 797.919,A 0.000,B 0.000,C 90.000,E1 345.463} C_DIS
LIN {X 0.014,Y -198.239,Z 797.896,A 0.000,B 0.000,C 90.000,E1 341.348} C_DIS
LIN {X 0.010,Y -203.656,Z 797.874,A 0.000,B 0.000,C 90.000,E1 337.305} C_DIS
LIN {X 0.027,Y -208.705,Z 797.856,A 0.000,B 0.000,C 90.000,E1 334.101} C_DIS
LIN {X 0.118,Y -215.928,Z 797.834,A 0.000,B 0.000,C 90.000,E1 330.127} C_DIS
LIN {X 0.008,Y -222.241,Z 797.817,A 0.000,B 0.000,C 90.000,E1 327.041} C_DIS
LIN {X -0.080,Y -229.004,Z 797.800,A 0.000,B 0.000,C 90.000,E1 323.989} C_DIS
LIN {X -0.025,Y -238.134,Z 797.779,A 0.000,B 0.000,C 90.000,E1 320.194} C_DIS
LIN {X -0.063,Y -247.173,Z 797.760,A 0.000,B 0.000,C 90.000,E1 316.863} C_DIS
LIN {X -0.015,Y -258.001,Z 797.740,A 0.000,B 0.000,C 90.000,E1 313.218} C_DIS
LIN {X -0.005,Y -268.551,Z 797.722,A 0.000,B 0.000,C 90.000,E1 310.011} C_DIS
LIN {X 0.118,Y -281.350,Z 797.703,A 0.000,B 0.000,C 90.000,E1 306.503} C_DIS
LIN {X 0.073,Y -294.056,Z 797.686,A 0.000,B 0.000,C 90.000,E1 303.452} C_DIS
LIN {X 0.044,Y -306.554,Z 797.671,A 0.000,B 0.000,C 90.000,E1 300.797} C_DIS
LIN {X -0.065,Y -318.584,Z 797.658,A 0.000,B 0.000,C 90.000,E1 298.537} C_DIS
LIN {X 0.001,Y -335.348,Z 797.643,A 0.000,B 0.000,C 90.000,E1 295.668} C_DIS
LIN {X -0.062,Y -351.408,Z 797.629,A 0.000,B 0.000,C 90.000,E1 293.206} C_DIS
LIN {X 0.003,Y -369.108,Z 797.615,A 0.000,B 0.000,C 90.000,E1 290.791} C_DIS
LIN {X -0.064,Y -391.085,Z 797.601,A 0.000,B 0.000,C 90.000,E1 288.181} C_DIS
LIN {X 0.136,Y -408.559,Z 797.590,A 0.000,B 0.000,C 90.000,E1 286.205} C_DIS
LIN {X -0.188,Y -420.880,Z 797.583,A 0.000,B 0.000,C 90.000,E1 284.898} C_DIS
LIN {X -0.138,Y -433.133,Z 797.575,A 0.000,B 0.000,C 90.000,E1 283.536} C_DIS
LIN {X -0.010,Y -445.029,Z 797.568,A 0.000,B 0.000,C 90.000,E1 282.187} C_DIS
LIN {X 0.052,Y -453.993,Z 797.562,A 0.000,B 0.000,C 90.000,E1 281.130} C_DIS
LIN {X 0.216,Y -462.241,Z 797.556,A 0.000,B 0.000,C 90.000,E1 280.074} C_DIS
LIN {X -0.143,Y -469.886,Z 797.550,A 0.000,B 0.000,C 90.000,E1 279.095} C_DIS
LIN {X -0.198,Y -475.161,Z 797.546,A 0.000,B 0.000,C 90.000,E1 278.341} C_DIS
LIN {X -0.213,Y -479.819,Z 797.542,A 0.000,B 0.000,C 90.000,E1 277.587} C_DIS
LIN {X -0.184,Y -483.847,Z 797.538,A 0.000,B 0.000,C 90.000,E1 276.834} C_DIS
LIN {X -0.181,Y -487.190,Z 797.534,A 0.000,B 0.000,C 90.000,E1 276.087} C_DIS
LIN {X 0.020,Y -488.997,Z 797.531,A 0.000,B 0.000,C 90.000,E1 275.568} C_DIS
LIN {X 0.228,Y -490.466,Z 797.528,A 0.000,B 0.000,C 90.000,E1 275.049} C_DIS
LIN {X -0.045,Y -491.540,Z 797.525,A 0.000,B 0.000,C 90.000,E1 274.588} C_DIS
LIN {X 0.143,Y -492.211,Z 797.523,A 0.000,B 0.000,C 90.000,E1 274.073} C_DIS
LIN {X -0.119,Y -492.494,Z 797.520,A 0.000,B 0.000,C 90.000,E1 273.612} C_DIS
LIN {X 0.111,Y -492.375,Z 797.517,A 0.000,B 0.000,C 90.000,E1 273.094} C_DIS
LIN {X -0.176,Y -491.828,Z 797.515,A 0.000,B 0.000,C 90.000,E1 272.636} C_DIS
LIN {X 0.031,Y -490.900,Z 797.512,A 0.000,B 0.000,C 90.000,E1 272.121} C_DIS
LIN {X -0.239,Y -489.531,Z 797.509,A 0.000,B 0.000,C 90.000,E1 271.661} C_DIS
LIN {X -0.040,Y -487.765,Z 797.506,A 0.000,B 0.000,C 90.000,E1 271.146} C_DIS
LIN {X 0.150,Y -485.475,Z 797.504,A 0.000,B 0.000,C 90.000,E1 270.630} C_DIS
LIN {X -0.159,Y -482.689,Z 797.501,A 0.000,B 0.000,C 90.000,E1 270.172} C_DIS
LIN {X 0.002,Y -479.305,Z 797.498,A 0.000,B 0.000,C 90.000,E1 269.656} C_DIS
LIN {X 0.141,Y -475.133,Z 797.495,A 0.000,B 0.000,C 90.000,E1 269.141} C_DIS
LIN {X -0.214,Y -470.011,Z 797.493,A 0.000,B 0.000,C 90.000,E1 268.682} C_DIS
LIN {X 0.159,Y -464.015,Z 797.490,A 0.000,B 0.000,C 90.000,E1 268.165} C_DIS
LIN {X 0.076,Y -457.316,Z 797.488,A 0.000,B 0.000,C 90.000,E1 267.764} C_DIS
LIN {X 0.123,Y -449.916,Z 797.486,A 0.000,B 0.000,C 90.000,E1 267.421} C_DIS
LIN {X -0.099,Y -442.349,Z 797.484,A 0.000,B 0.000,C 90.000,E1 267.192} C_DIS
LIN {X 0.157,Y -434.242,Z 797.483,A 0.000,B 0.000,C 90.000,E1 266.963} C_DIS
LIN {X -0.181,Y -426.860,Z 797.483,A 0.000,B 0.000,C 90.000,E1 266.906} C_DIS
LIN {X -0.108,Y -418.868,Z 797.482,A 0.000,B 0.000,C 90.000,E1 266.846} C_DIS
LIN {X -0.073,Y -180.974,Z 797.482,A 0.000,B 0.000,C 90.000,E1 266.846} C_DIS
LIN {X -0.085,Y -180.880,Z 797.473,A 0.000,B 0.000,C 90.000,E1 265.122} C_DIS
LIN {X -0.025,Y -179.000,Z 797.445,A 0.000,B 0.000,C 90.000,E1 260.038} C_DIS
LIN {X 0.070,Y -178.595,Z 797.440,A 0.000,B 0.000,C 90.000,E1 259.162} C_DIS
LIN {X -0.037,Y -175.648,Z 797.412,A 0.000,B 0.000,C 90.000,E1 254.102} C_DIS
LIN {X -0.032,Y -172.367,Z 797.388,A 0.000,B 0.000,C 90.000,E1 249.826} C_DIS
LIN {X -0.017,Y -171.156,Z 797.378,A 0.000,B 0.000,C 90.000,E1 248.103} C_DIS
LIN {X 0.027,Y -167.457,Z 797.354,A 0.000,B 0.000,C 90.000,E1 243.768} C_DIS
LIN {X -0.039,Y -166.853,Z 797.349,A 0.000,B 0.000,C 90.000,E1 242.922} C_DIS
LIN {X 0.025,Y -162.838,Z 797.325,A 0.000,B 0.000,C 90.000,E1 238.535} C_DIS
LIN {X 0.000,Y -161.522,Z 797.315,A 0.000,B 0.000,C 90.000,E1 236.786} C_DIS
LIN {X 0.041,Y -157.521,Z 797.291,A 0.000,B 0.000,C 90.000,E1 232.351} C_DIS
LIN {X -0.026,Y -155.546,Z 797.276,A 0.000,B 0.000,C 90.000,E1 229.703} C_DIS
LIN {X 0.016,Y -151.838,Z 797.251,A 0.000,B 0.000,C 90.000,E1 225.202} C_DIS
LIN {X -0.077,Y -150.056,Z 797.236,A 0.000,B 0.000,C 90.000,E1 222.528} C_DIS
LIN {X 0.048,Y -146.868,Z 797.211,A 0.000,B 0.000,C 90.000,E1 217.935} C_DIS
LIN {X -0.053,Y -145.452,Z 797.196,A 0.000,B 0.000,C 90.000,E1 215.231} C_DIS
LIN {X 0.061,Y -142.869,Z 797.170,A 0.000,B 0.000,C 90.000,E1 210.590} C_DIS
LIN {X -0.014,Y -141.486,Z 797.150,A 0.000,B 0.000,C 90.000,E1 206.924} C_DIS
LIN {X -0.028,Y -139.383,Z 797.113,A 0.000,B 0.000,C 90.000,E1 200.429} C_DIS
LIN {X -0.040,Y -138.839,Z 797.098,A 0.000,B 0.000,C 90.000,E1 197.638} C_DIS
LIN {X 0.021,Y -138.354,Z 797.056,A 0.000,B 0.000,C 90.000,E1 190.141} C_DIS
LIN {X 0.016,Y -139.522,Z 797.005,A 0.000,B 0.000,C 90.000,E1 180.802} C_DIS
LIN {X -0.044,Y -141.185,Z 796.973,A 0.000,B 0.000,C 90.000,E1 175.241} C_DIS
LIN {X 0.069,Y -142.563,Z 796.958,A 0.000,B 0.000,C 90.000,E1 172.413} C_DIS
LIN {X 0.024,Y -144.847,Z 796.932,A 0.000,B 0.000,C 90.000,E1 167.813} C_DIS
LIN {X -0.020,Y -147.472,Z 796.912,A 0.000,B 0.000,C 90.000,E1 164.157} C_DIS
LIN {X 0.006,Y -150.056,Z 796.892,A 0.000,B 0.000,C 90.000,E1 160.496} C_DIS
LIN {X 0.011,Y -153.401,Z 796.872,A 0.000,B 0.000,C 90.000,E1 156.869} C_DIS
LIN {X 0.057,Y -155.931,Z 796.857,A 0.000,B 0.000,C 90.000,E1 154.152} C_DIS
LIN {X 0.031,Y -159.800,Z 796.837,A 0.000,B 0.000,C 90.000,E1 150.589} C_DIS
LIN {X 0.016,Y -162.040,Z 796.827,A 0.000,B 0.000,C 90.000,E1 148.820} C_DIS
LIN {X -0.010,Y -166.235,Z 796.807,A 0.000,B 0.000,C 90.000,E1 145.308} C_DIS
LIN {X -0.009,Y -171.251,Z 796.788,A 0.000,B 0.000,C 90.000,E1 141.823} C_DIS
LIN {X -0.086,Y -176.141,Z 796.769,A 0.000,B 0.000,C 90.000,E1 138.405} C_DIS
LIN {X 0.030,Y -180.409,Z 796.755,A 0.000,B 0.000,C 90.000,E1 135.810} C_DIS
LIN {X 0.006,Y -185.815,Z 796.736,A 0.000,B 0.000,C 90.000,E1 132.447} C_DIS
LIN {X 0.060,Y -190.435,Z 796.722,A 0.000,B 0.000,C 90.000,E1 129.930} C_DIS
LIN {X -0.015,Y -192.600,Z 796.715,A 0.000,B 0.000,C 90.000,E1 128.669} C_DIS
LIN {X -0.053,Y -292.760,Z 796.715,A 0.000,B 0.000,C 90.000,E1 128.669} C_DIS
LIN {X -0.036,Y -294.862,Z 796.715,A 0.000,B 0.000,C 90.000,E1 128.624} C_DIS
LIN {X -0.033,Y -300.377,Z 796.713,A 0.000,B 0.000,C 90.000,E1 128.302} C_DIS
LIN {X 0.019,Y -303.584,Z 796.711,A 0.000,B 0.000,C 90.000,E1 127.935} C_DIS
LIN {X -0.091,Y -305.561,Z 796.709,A 0.000,B 0.000,C 90.000,E1 127.649} C_DIS
LIN {X 0.042,Y -307.108,Z 796.707,A 0.000,B 0.000,C 90.000,E1 127.317} C_DIS
LIN {X 0.007,Y -308.416,Z 796.706,A 0.000,B 0.000,C 90.000,E1 126.996} C_DIS
LIN {X 0.128,Y -320.511,Z 796.684,A 0.000,B 0.000,C 90.000,E1 123.086} C_DIS
LIN {X -0.028,Y -330.958,Z 796.668,A 0.000,B 0.000,C 90.000,E1 120.256} C_DIS
LIN {X -0.092,Y -342.757,Z 796.652,A 0.000,B 0.000,C 90.000,E1 117.462} C_DIS
LIN {X 0.022,Y -356.021,Z 796.637,A 0.000,B 0.000,C 90.000,E1 114.695} C_DIS
LIN {X -0.168,Y -369.129,Z 796.624,A 0.000,B 0.000,C 90.000,E1 112.333} C_DIS
LIN {X 0.189,Y -383.579,Z 796.611,A 0.000,B 0.000,C 90.000,E1 109.939} C_DIS
LIN {X -0.077,Y -399.473,Z 796.598,A 0.000,B 0.000,C 90.000,E1 107.692} C_DIS
LIN {X 0.187,Y -416.926,Z 796.586,A 0.000,B 0.000,C 90.000,E1 105.426} C_DIS
LIN {X -0.130,Y -436.054,Z 796.574,A 0.000,B 0.000,C 90.000,E1 103.300} C_DIS
LIN {X 0.079,Y -456.181,Z 796.563,A 0.000,B 0.000,C 90.000,E1 101.243} C_DIS
LIN {X -0.070,Y -466.453,Z 796.557,A 0.000,B 0.000,C 90.000,E1 100.310} C_DIS
LIN {X -0.027,Y -468.813,Z 796.556,A 0.000,B 0.000,C 90.000,E1 100.074} C_DIS
LIN {X -0.063,Y -470.601,Z 796.555,A 0.000,B 0.000,C 90.000,E1 99.849} C_DIS
LIN {X -0.212,Y -472.099,Z 796.553,A 0.000,B 0.000,C 90.000,E1 99.613} C_DIS
LIN {X 0.104,Y -473.217,Z 796.552,A 0.000,B 0.000,C 90.000,E1 99.321} C_DIS
LIN {X 0.215,Y -474.549,Z 796.549,A 0.000,B 0.000,C 90.000,E1 98.803} C_DIS
LIN {X -0.134,Y -474.864,Z 796.546,A 0.000,B 0.000,C 90.000,E1 98.341} C_DIS
LIN {X 0.061,Y -474.215,Z 796.543,A 0.000,B 0.000,C 90.000,E1 97.814} C_DIS
LIN {X 0.190,Y -472.500,Z 796.541,A 0.000,B 0.000,C 90.000,E1 97.296} C_DIS
LIN {X -0.011,Y -471.148,Z 796.539,A 0.000,B 0.000,C 90.000,E1 97.068} C_DIS
LIN {X -0.072,Y -454.910,Z 796.525,A 0.000,B 0.000,C 90.000,E1 94.531} C_DIS
LIN {X 0.028,Y -441.344,Z 796.512,A 0.000,B 0.000,C 90.000,E1 92.178} C_DIS
LIN {X 0.181,Y -432.054,Z 796.503,A 0.000,B 0.000,C 90.000,E1 90.573} C_DIS
LIN {X -0.147,Y -420.944,Z 796.493,A 0.000,B 0.000,C 90.000,E1 88.740} C_DIS
LIN {X 0.170,Y -409.606,Z 796.482,A 0.000,B 0.000,C 90.000,E1 86.788} C_DIS
LIN {X -0.157,Y -398.132,Z 796.471,A 0.000,B 0.000,C 90.000,E1 84.894} C_DIS
LIN {X 0.177,Y -383.587,Z 796.457,A 0.000,B 0.000,C 90.000,E1 82.299} C_DIS
LIN {X -0.158,Y -369.492,Z 796.443,A 0.000,B 0.000,C 90.000,E1 79.746} C_DIS
LIN {X 0.025,Y -354.473,Z 796.426,A 0.000,B 0.000,C 90.000,E1 76.756} C_DIS
LIN {X 0.004,Y -342.863,Z 796.413,A 0.000,B 0.000,C 90.000,E1 74.338} C_DIS
LIN {X -0.020,Y -331.389,Z 796.399,A 0.000,B 0.000,C 90.000,E1 71.873} C_DIS
LIN {X 0.089,Y -320.168,Z 796.385,A 0.000,B 0.000,C 90.000,E1 69.337} C_DIS
LIN {X 0.098,Y -305.414,Z 796.366,A 0.000,B 0.000,C 90.000,E1 65.793} C_DIS
LIN {X 0.132,Y -293.097,Z 796.347,A 0.000,B 0.000,C 90.000,E1 62.487} C_DIS
LIN {X 0.108,Y -282.671,Z 796.330,A 0.000,B 0.000,C 90.000,E1 59.459} C_DIS
LIN {X -0.129,Y -272.861,Z 796.313,A 0.000,B 0.000,C 90.000,E1 56.421} C_DIS
LIN {X -0.082,Y -264.454,Z 796.298,A 0.000,B 0.000,C 90.000,E1 53.623} C_DIS
LIN {X -0.145,Y -256.090,Z 796.282,A 0.000,B 0.000,C 90.000,E1 50.803} C_DIS
LIN {X 0.060,Y -247.915,Z 796.266,A 0.000,B 0.000,C 90.000,E1 47.877} C_DIS
LIN {X 0.142,Y -238.320,Z 796.246,A 0.000,B 0.000,C 90.000,E1 44.190} C_DIS
LIN {X 0.043,Y -231.077,Z 796.229,A 0.000,B 0.000,C 90.000,E1 41.229} C_DIS
LIN {X -0.041,Y -224.059,Z 796.212,A 0.000,B 0.000,C 90.000,E1 38.222} C_DIS
LIN {X 0.018,Y -215.658,Z 796.191,A 0.000,B 0.000,C 90.000,E1 34.358} C_DIS
LIN {X -0.085,Y -209.473,Z 796.174,A 0.000,B 0.000,C 90.000,E1 31.258} C_DIS
LIN {X 0.051,Y -203.993,Z 796.156,A 0.000,B 0.000,C 90.000,E1 28.052} C_DIS
LIN {X 0.046,Y -199.232,Z 796.138,A 0.000,B 0.000,C 90.000,E1 24.847} C_DIS
LIN {X 0.055,Y -194.277,Z 796.116,A 0.000,B 0.000,C 90.000,E1 20.791} C_DIS
LIN {X -0.072,Y -190.454,Z 796.093,A 0.000,B 0.000,C 90.000,E1 16.732} C_DIS
LIN {X -0.061,Y -187.366,Z 796.065,A 0.000,B 0.000,C 90.000,E1 11.771} C_DIS
LIN {X 0.046,Y -185.466,Z 796.014,A 0.000,B 0.000,C 90.000,E1 2.579} C_DIS
LIN {X -0.039,Y -187.539,Z 795.970,A 0.000,B 0.000,C 90.000,E1 354.546} C_DIS
LIN {X -0.023,Y -190.532,Z 795.942,A 0.000,B 0.000,C 90.000,E1 349.567} C_DIS
LIN {X -0.070,Y -193.991,Z 795.919,A 0.000,B 0.000,C 90.000,E1 345.463} C_DIS
LIN {X 0.038,Y -198.375,Z 795.896,A 0.000,B 0.000,C 90.000,E1 341.348} C_DIS
LIN {X 0.038,Y -203.818,Z 795.874,A 0.000,B 0.000,C 90.000,E1 337.305} C_DIS
LIN {X 0.060,Y -208.877,Z 795.856,A 0.000,B 0.000,C 90.000,E1 334.101} C_DIS
LIN {X -0.029,Y -216.080,Z 795.834,A 0.000,B 0.000,C 90.000,E1 330.177} C_DIS
LIN {X 0.054,Y -222.397,Z 795.817,A 0.000,B 0.000,C 90.000,E1 327.041} C_DIS
LIN {X 0.041,Y -230.909,Z 795.796,A 0.000,B 0.000,C 90.000,E1 323.210} C_DIS
LIN {X -0.027,Y -240.191,Z 795.775,A 0.000,B 0.000,C 90.000,E1 319.461} C_DIS
LIN {X 0.155,Y -250.429,Z 795.754,A 0.000,B 0.000,C 90.000,E1 315.729} C_DIS
LIN {X -0.072,Y -260.338,Z 795.736,A 0.000,B 0.000,C 90.000,E1 312.528} C_DIS
LIN {X -0.088,Y -272.271,Z 795.716,A 0.000,B 0.000,C 90.000,E1 308.991} C_DIS
LIN {X -0.014,Y -285.424,Z 795.697,A 0.000,B 0.000,C 90.000,E1 305.518} C_DIS
LIN {X 0.048,Y -298.541,Z 795.680,A 0.000,B 0.000,C 90.000,E1 302.467} C_DIS
LIN {X -0.192,Y -311.500,Z 795.666,A 0.000,B 0.000,C 90.000,E1 299.873} C_DIS
LIN {X 0.055,Y -329.525,Z 795.648,A 0.000,B 0.000,C 90.000,E1 296.616} C_DIS
LIN {X 0.004,Y -349.165,Z 795.631,A 0.000,B 0.000,C 90.000,E1 293.515} C_DIS
LIN {X 0.089,Y -368.905,Z 795.616,A 0.000,B 0.000,C 90.000,E1 290.791} C_DIS
LIN {X -0.004,Y -390.865,Z 795.601,A 0.000,B 0.000,C 90.000,E1 288.181} C_DIS
LIN {X 0.031,Y -405.896,Z 795.592,A 0.000,B 0.000,C 90.000,E1 286.496} C_DIS
LIN {X -0.117,Y -418.444,Z 795.584,A 0.000,B 0.000,C 90.000,E1 285.134} C_DIS
LIN {X -0.103,Y -430.745,Z 795.576,A 0.000,B 0.000,C 90.000,E1 283.772} C_DIS
LIN {X 0.093,Y -442.690,Z 795.569,A 0.000,B 0.000,C 90.000,E1 282.411} C_DIS
LIN {X 0.033,Y -451.770,Z 795.563,A 0.000,B 0.000,C 90.000,E1 281.366} C_DIS
LIN {X 0.172,Y -460.206,Z 795.557,A 0.000,B 0.000,C 90.000,E1 280.310} C_DIS
LIN {X -0.133,Y -467.984,Z 795.552,A 0.000,B 0.000,C 90.000,E1 279.321} C_DIS
LIN {X -0.213,Y -473.368,Z 795.547,A 0.000,B 0.000,C 90.000,E1 278.568} C_DIS
LIN {X 0.232,Y -478.289,Z 795.543,A 0.000,B 0.000,C 90.000,E1 277.757} C_DIS
LIN {X 0.185,Y -482.562,Z 795.539,A 0.000,B 0.000,C 90.000,E1 277.011} C_DIS
LIN {X 0.240,Y -486.153,Z 795.535,A 0.000,B 0.000,C 90.000,E1 276.258} C_DIS
LIN {X -0.219,Y -488.973,Z 795.531,A 0.000,B 0.000,C 90.000,E1 275.568} C_DIS
LIN {X -0.012,Y -490.427,Z 795.528,A 0.000,B 0.000,C 90.000,E1 275.049} C_DIS
LIN {X 0.205,Y -491.528,Z 795.525,A 0.000,B 0.000,C 90.000,E1 274.531} C_DIS
LIN {X -0.099,Y -492.196,Z 795.523,A 0.000,B 0.000,C 90.000,E1 274.073} C_DIS
LIN {X 0.131,Y -492.494,Z 795.520,A 0.000,B 0.000,C 90.000,E1 273.555} C_DIS
LIN {X -0.130,Y -492.340,Z 795.517,A 0.000,B 0.000,C 90.000,E1 273.094} C_DIS
LIN {X 0.074,Y -491.811,Z 795.514,A 0.000,B 0.000,C 90.000,E1 272.579} C_DIS
LIN {X -0.209,Y -490.853,Z 795.512,A 0.000,B 0.000,C 90.000,E1 272.121} C_DIS
LIN {X 0.010,Y -489.500,Z 795.509,A 0.000,B 0.000,C 90.000,E1 271.604} C_DIS
LIN {X 0.059,Y -486.644,Z 795.505,A 0.000,B 0.000,C 90.000,E1 270.859} C_DIS
LIN {X 0.241,Y -484.107,Z 795.502,A 0.000,B 0.000,C 90.000,E1 270.344} C_DIS
LIN {X -0.075,Y -481.028,Z 795.499,A 0.000,B 0.000,C 90.000,E1 269.885} C_DIS
LIN {X 0.075,Y -477.200,Z 795.497,A 0.000,B 0.000,C 90.000,E1 269.370} C_DIS
LIN {X 0.202,Y -472.595,Z 795.494,A 0.000,B 0.000,C 90.000,E1 268.854} C_DIS
LIN {X 0.004,Y -467.092,Z 795.491,A 0.000,B 0.000,C 90.000,E1 268.396} C_DIS
LIN {X -0.001,Y -464.004,Z 795.490,A 0.000,B 0.000,C 90.000,E1 268.165} C_DIS
LIN {X -0.068,Y -457.307,Z 795.488,A 0.000,B 0.000,C 90.000,E1 267.764} C_DIS
LIN {X 0.001,Y -450.046,Z 795.486,A 0.000,B 0.000,C 90.000,E1 267.421} C_DIS
LIN {X 0.195,Y -442.396,Z 795.484,A 0.000,B 0.000,C 90.000,E1 267.135} C_DIS
LIN {X -0.001,Y -434.077,Z 795.483,A 0.000,B 0.000,C 90.000,E1 266.963} C_DIS
LIN {X 0.103,Y -426.775,Z 795.483,A 0.000,B 0.000,C 90.000,E1 266.849} C_DIS
LIN {X 0.179,Y -419.401,Z 795.482,A 0.000,B 0.000,C 90.000,E1 266.788} C_DIS
LIN {X 0.051,Y -180.973,Z 795.482,A 0.000,B 0.000,C 90.000,E1 266.788} C_DIS
LIN {X 0.041,Y -180.878,Z 795.473,A 0.000,B 0.000,C 90.000,E1 265.065} C_DIS
LIN {X -0.079,Y -178.996,Z 795.445,A 0.000,B 0.000,C 90.000,E1 260.038} C_DIS
LIN {X 0.015,Y -178.582,Z 795.440,A 0.000,B 0.000,C 90.000,E1 259.162} C_DIS
LIN {X -0.091,Y -175.635,Z 795.411,A 0.000,B 0.000,C 90.000,E1 254.102} C_DIS
LIN {X -0.024,Y -172.355,Z 795.388,A 0.000,B 0.000,C 90.000,E1 249.806} C_DIS
LIN {X -0.070,Y -171.139,Z 795.378,A 0.000,B 0.000,C 90.000,E1 248.103} C_DIS
LIN {X -0.025,Y -167.444,Z 795.354,A 0.000,B 0.000,C 90.000,E1 243.768} C_DIS
LIN {X 0.057,Y -166.840,Z 795.349,A 0.000,B 0.000,C 90.000,E1 242.871} C_DIS
LIN {X -0.026,Y -162.824,Z 795.325,A 0.000,B 0.000,C 90.000,E1 238.535} C_DIS
LIN {X 0.038,Y -161.508,Z 795.315,A 0.000,B 0.000,C 90.000,E1 236.755} C_DIS
LIN {X -0.010,Y -157.507,Z 795.291,A 0.000,B 0.000,C 90.000,E1 232.351} C_DIS
LIN {X 0.024,Y -155.529,Z 795.276,A 0.000,B 0.000,C 90.000,E1 229.666} C_DIS
LIN {X 0.074,Y -151.825,Z 795.251,A 0.000,B 0.000,C 90.000,E1 225.162} C_DIS
LIN {X 0.086,Y -150.040,Z 795.236,A 0.000,B 0.000,C 90.000,E1 222.447} C_DIS
LIN {X 0.000,Y -146.857,Z 795.211,A 0.000,B 0.000,C 90.000,E1 217.935} C_DIS
LIN {X 0.018,Y -145.440,Z 795.195,A 0.000,B 0.000,C 90.000,E1 215.185} C_DIS
LIN {X 0.013,Y -142.861,Z 795.170,A 0.000,B 0.000,C 90.000,E1 210.590} C_DIS
LIN {X 0.065,Y -141.477,Z 795.149,A 0.000,B 0.000,C 90.000,E1 206.873} C_DIS
LIN {X -0.075,Y -139.381,Z 795.113,A 0.000,B 0.000,C 90.000,E1 200.429} C_DIS
LIN {X 0.046,Y -138.834,Z 795.098,A 0.000,B 0.000,C 90.000,E1 197.583} C_DIS
LIN {X -0.026,Y -138.354,Z 795.056,A 0.000,B 0.000,C 90.000,E1 190.141} C_DIS
LIN {X -0.031,Y -139.524,Z 795.004,A 0.000,B 0.000,C 90.000,E1 180.802} C_DIS
LIN {X 0.062,Y -141.193,Z 794.973,A 0.000,B 0.000,C 90.000,E1 175.179} C_DIS
LIN {X 0.021,Y -142.570,Z 794.958,A 0.000,B 0.000,C 90.000,E1 172.413} C_DIS
LIN {X -0.024,Y -144.859,Z 794.932,A 0.000,B 0.000,C 90.000,E1 167.813} C_DIS
LIN {X -0.069,Y -147.484,Z 794.912,A 0.000,B 0.000,C 90.000,E1 164.157} C_DIS
LIN {X -0.043,Y -150.071,Z 794.892,A 0.000,B 0.000,C 90.000,E1 160.496} C_DIS
LIN {X -0.039,Y -153.420,Z 794.871,A 0.000,B 0.000,C 90.000,E1 156.869} C_DIS
LIN {X 0.009,Y -156.840,Z 794.851,A 0.000,B 0.000,C 90.000,E1 153.256} C_DIS
LIN {X 0.080,Y -160.920,Z 794.832,A 0.000,B 0.000,C 90.000,E1 149.665} C_DIS
LIN {X 0.025,Y -163.045,Z 794.822,A 0.000,B 0.000,C 90.000,E1 147.916} C_DIS
LIN {X 0.030,Y -167.437,Z 794.802,A 0.000,B 0.000,C 90.000,E1 144.402} C_DIS
LIN {X -0.061,Y -171.276,Z 794.788,A 0.000,B 0.000,C 90.000,E1 141.823} C_DIS
LIN {X -0.022,Y -176.168,Z 794.769,A 0.000,B 0.000,C 90.000,E1 138.366} C_DIS
LIN {X -0.025,Y -180.440,Z 794.754,A 0.000,B 0.000,C 90.000,E1 135.810} C_DIS
LIN {X -0.050,Y -185.845,Z 794.736,A 0.000,B 0.000,C 90.000,E1 132.447} C_DIS
LIN {X 0.004,Y -190.468,Z 794.722,A 0.000,B 0.000,C 90.000,E1 129.930} C_DIS
LIN {X 0.020,Y -192.582,Z 794.715,A 0.000,B 0.000,C 90.000,E1 128.669} C_DIS
LIN {X -0.003,Y -292.178,Z 794.715,A 0.000,B 0.000,C 90.000,E1 128.669} C_DIS
LIN {X -0.107,Y -293.830,Z 794.715,A 0.000,B 0.000,C 90.000,E1 128.669} C_DIS
LIN {X 0.003,Y -298.229,Z 794.714,A 0.000,B 0.000,C 90.000,E1 128.463} C_DIS
LIN {X 0.115,Y -300.591,Z 794.713,A 0.000,B 0.000,C 90.000,E1 128.257} C_DIS
LIN {X 0.034,Y -304.438,Z 794.710,A 0.000,B 0.000,C 90.000,E1 127.810} C_DIS
LIN {X -0.170,Y -306.306,Z 794.708,A 0.000,B 0.000,C 90.000,E1 127.523} C_DIS
LIN {X 0.055,Y -307.764,Z 794.706,A 0.000,B 0.000,C 90.000,E1 127.156} C_DIS
LIN {X 0.049,Y -309.868,Z 794.703,A 0.000,B 0.000,C 90.000,E1 126.503} C_DIS
LIN {X -0.093,Y -319.925,Z 794.685,A 0.000,B 0.000,C 90.000,E1 123.293} C_DIS
LIN {X 0.015,Y -330.294,Z 794.669,A 0.000,B 0.000,C 90.000,E1 120.413} C_DIS
LIN {X 0.102,Y -342.016,Z 794.653,A 0.000,B 0.000,C 90.000,E1 117.590} C_DIS
LIN {X 0.057,Y -355.187,Z 794.638,A 0.000,B 0.000,C 90.000,E1 114.847} C_DIS
LIN {X 0.003,Y -368.211,Z 794.625,A 0.000,B 0.000,C 90.000,E1 112.461} C_DIS
LIN {X -0.014,Y -382.570,Z 794.612,A 0.000,B 0.000,C 90.000,E1 110.120} C_DIS
LIN {X 0.066,Y -398.365,Z 794.599,A 0.000,B 0.000,C 90.000,E1 107.819} C_DIS
LIN {X -0.086,Y -415.713,Z 794.587,A 0.000,B 0.000,C 90.000,E1 105.607} C_DIS
LIN {X 0.083,Y -434.723,Z 794.575,A 0.000,B 0.000,C 90.000,E1 103.411} C_DIS
LIN {X 0.113,Y -454.813,Z 794.563,A 0.000,B 0.000,C 90.000,E1 101.366} C_DIS
LIN {X -0.061,Y -467.647,Z 794.557,A 0.000,B 0.000,C 90.000,E1 100.197} C_DIS
LIN {X -0.043,Y -469.745,Z 794.555,A 0.000,B 0.000,C 90.000,E1 99.962} C_DIS
LIN {X -0.026,Y -471.338,Z 794.554,A 0.000,B 0.000,C 90.000,E1 99.726} C_DIS
LIN {X -0.251,Y -472.651,Z 794.553,A 0.000,B 0.000,C 90.000,E1 99.500} C_DIS
LIN {X 0.068,Y -473.621,Z 794.551,A 0.000,B 0.000,C 90.000,E1 99.208} C_DIS
LIN {X 0.184,Y -474.710,Z 794.548,A 0.000,B 0.000,C 90.000,E1 98.690} C_DIS
LIN {X -0.094,Y -474.808,Z 794.546,A 0.000,B 0.000,C 90.000,E1 98.219} C_DIS
LIN {X 0.035,Y -473.933,Z 794.543,A 0.000,B 0.000,C 90.000,E1 97.701} C_DIS
LIN {X 0.164,Y -471.942,Z 794.540,A 0.000,B 0.000,C 90.000,E1 97.182} C_DIS
LIN {X -0.072,Y -465.401,Z 794.534,A 0.000,B 0.000,C 90.000,E1 96.201} C_DIS
LIN {X 0.116,Y -449.646,Z 794.520,A 0.000,B 0.000,C 90.000,E1 93.612} C_DIS
LIN {X 0.166,Y -439.143,Z 794.510,A 0.000,B 0.000,C 90.000,E1 91.776} C_DIS
LIN {X -0.166,Y -429.791,Z 794.501,A 0.000,B 0.000,C 90.000,E1 90.229} C_DIS
LIN {X -0.106,Y -418.616,Z 794.491,A 0.000,B 0.000,C 90.000,E1 88.339} C_DIS
LIN {X 0.152,Y -407.276,Z 794.480,A 0.000,B 0.000,C 90.000,E1 86.388} C_DIS
LIN {X 0.208,Y -395.788,Z 794.469,A 0.000,B 0.000,C 90.000,E1 84.432} C_DIS
LIN {X 0.085,Y -381.337,Z 794.455,A 0.000,B 0.000,C 90.000,E1 81.894} C_DIS
LIN {X 0.065,Y -368.861,Z 794.442,A 0.000,B 0.000,C 90.000,E1 79.577} C_DIS
LIN {X -0.186,Y -352.439,Z 794.424,A 0.000,B 0.000,C 90.000,E1 76.353} C_DIS
LIN {X -0.166,Y -340.867,Z 794.411,A 0.000,B 0.000,C 90.000,E1 73.921} C_DIS
LIN {X 0.079,Y -329.453,Z 794.397,A 0.000,B 0.000,C 90.000,E1 71.402} C_DIS
LIN {X -0.059,Y -318.284,Z 794.383,A 0.000,B 0.000,C 90.000,E1 68.901} C_DIS
LIN {X -0.005,Y -304.984,Z 794.365,A 0.000,B 0.000,C 90.000,E1 65.665} C_DIS
LIN {X 0.021,Y -292.769,Z 794.346,A 0.000,B 0.000,C 90.000,E1 62.359} C_DIS
LIN {X -0.040,Y -281.312,Z 794.328,A 0.000,B 0.000,C 90.000,E1 58.997} C_DIS
LIN {X 0.127,Y -272.668,Z 794.312,A 0.000,B 0.000,C 90.000,E1 56.215} C_DIS
LIN {X 0.161,Y -264.314,Z 794.297,A 0.000,B 0.000,C 90.000,E1 53.417} C_DIS
LIN {X 0.084,Y -255.998,Z 794.281,A 0.000,B 0.000,C 90.000,E1 50.598} C_DIS
LIN {X 0.088,Y -247.857,Z 794.265,A 0.000,B 0.000,C 90.000,E1 47.715} C_DIS
LIN {X -0.001,Y -238.298,Z 794.245,A 0.000,B 0.000,C 90.000,E1 44.069} C_DIS
LIN {X 0.068,Y -231.054,Z 794.228,A 0.000,B 0.000,C 90.000,E1 41.067} C_DIS
LIN {X 0.018,Y -224.044,Z 794.211,A 0.000,B 0.000,C 90.000,E1 38.051} C_DIS
LIN {X 0.032,Y -215.663,Z 794.190,A 0.000,B 0.000,C 90.000,E1 34.199} C_DIS
LIN {X -0.007,Y -209.516,Z 794.173,A 0.000,B 0.000,C 90.000,E1 31.082} C_DIS
LIN {X 0.050,Y -204.043,Z 794.155,A 0.000,B 0.000,C 90.000,E1 27.897} C_DIS
LIN {X -0.047,Y -199.316,Z 794.137,A 0.000,B 0.000,C 90.000,E1 24.719} C_DIS
LIN {X -0.035,Y -194.398,Z 794.115,A 0.000,B 0.000,C 90.000,E1 20.663} C_DIS
LIN {X 0.021,Y -190.591,Z 794.092,A 0.000,B 0.000,C 90.000,E1 16.551} C_DIS
LIN {X 0.032,Y -187.536,Z 794.064,A 0.000,B 0.000,C 90.000,E1 11.591} C_DIS
LIN {X -0.060,Y -185.680,Z 794.014,A 0.000,B 0.000,C 90.000,E1 2.465} C_DIS
LIN {X -0.032,Y -187.717,Z 793.970,A 0.000,B 0.000,C 90.000,E1 354.546} C_DIS
LIN {X -0.009,Y -190.687,Z 793.942,A 0.000,B 0.000,C 90.000,E1 349.567} C_DIS
LIN {X -0.052,Y -194.137,Z 793.919,A 0.000,B 0.000,C 90.000,E1 345.463} C_DIS
LIN {X 0.061,Y -198.512,Z 793.896,A 0.000,B 0.000,C 90.000,E1 341.348} C_DIS
LIN {X 0.067,Y -203.975,Z 793.874,A 0.000,B 0.000,C 90.000,E1 337.305} C_DIS
LIN {X -0.094,Y -209.045,Z 793.856,A 0.000,B 0.000,C 90.000,E1 334.152} C_DIS
LIN {X -0.096,Y -216.229,Z 793.834,A 0.000,B 0.000,C 90.000,E1 330.205} C_DIS
LIN {X 0.099,Y -222.537,Z 793.817,A 0.000,B 0.000,C 90.000,E1 327.041} C_DIS
LIN {X 0.093,Y -231.046,Z 793.796,A 0.000,B 0.000,C 90.000,E1 323.210} C_DIS
LIN {X 0.031,Y -240.308,Z 793.775,A 0.000,B 0.000,C 90.000,E1 319.461} C_DIS
LIN {X 0.046,Y -249.448,Z 793.756,A 0.000,B 0.000,C 90.000,E1 316.134} C_DIS
LIN {X -0.004,Y -260.371,Z 793.736,A 0.000,B 0.000,C 90.000,E1 312.528} C_DIS
LIN {X -0.016,Y -272.286,Z 793.717,A 0.000,B 0.000,C 90.000,E1 308.991} C_DIS
LIN {X 0.061,Y -285.417,Z 793.697,A 0.000,B 0.000,C 90.000,E1 305.518} C_DIS
LIN {X -0.034,Y -298.491,Z 793.680,A 0.000,B 0.000,C 90.000,E1 302.498} C_DIS
LIN {X -0.113,Y -311.442,Z 793.666,A 0.000,B 0.000,C 90.000,E1 299.873} C_DIS
LIN {X 0.045,Y -327.564,Z 793.650,A 0.000,B 0.000,C 90.000,E1 296.950} C_DIS
LIN {X 0.079,Y -346.970,Z 793.632,A 0.000,B 0.000,C 90.000,E1 293.823} C_DIS
LIN {X 0.032,Y -364.168,Z 793.619,A 0.000,B 0.000,C 90.000,E1 291.408} C_DIS
LIN {X 0.063,Y -378.180,Z 793.609,A 0.000,B 0.000,C 90.000,E1 289.631} C_DIS
LIN {X -0.075,Y -395.574,Z 793.598,A 0.000,B 0.000,C 90.000,E1 287.638} C_DIS
LIN {X -0.071,Y -410.737,Z 793.589,A 0.000,B 0.000,C 90.000,E1 285.953} C_DIS
LIN {X -0.169,Y -423.214,Z 793.581,A 0.000,B 0.000,C 90.000,E1 284.592} C_DIS
LIN {X -0.099,Y -435.347,Z 793.573,A 0.000,B 0.000,C 90.000,E1 283.231} C_DIS
LIN {X -0.161,Y -444.800,Z 793.568,A 0.000,B 0.000,C 90.000,E1 282.175} C_DIS
LIN {X -0.201,Y -453.733,Z 793.562,A 0.000,B 0.000,C 90.000,E1 281.130} C_DIS
LIN {X -0.046,Y -461.975,Z 793.556,A 0.000,B 0.000,C 90.000,E1 280.074} C_DIS
LIN {X 0.126,Y -469.602,Z 793.550,A 0.000,B 0.000,C 90.000,E1 279.029} C_DIS
LIN {X 0.067,Y -474.870,Z 793.546,A 0.000,B 0.000,C 90.000,E1 278.276} C_DIS
LIN {X -0.015,Y -479.613,Z 793.542,A 0.000,B 0.000,C 90.000,E1 277.530} C_DIS
LIN {X 0.012,Y -483.696,Z 793.538,A 0.000,B 0.000,C 90.000,E1 276.777} C_DIS
LIN {X 0.016,Y -487.073,Z 793.534,A 0.000,B 0.000,C 90.000,E1 276.030} C_DIS
LIN {X 0.219,Y -488.868,Z 793.531,A 0.000,B 0.000,C 90.000,E1 275.511} C_DIS
LIN {X -0.062,Y -490.358,Z 793.528,A 0.000,B 0.000,C 90.000,E1 275.049} C_DIS
LIN {X 0.154,Y -491.479,Z 793.525,A 0.000,B 0.000,C 90.000,E1 274.531} C_DIS
LIN {X -0.149,Y -492.161,Z 793.523,A 0.000,B 0.000,C 90.000,E1 274.073} C_DIS
LIN {X 0.080,Y -492.447,Z 793.520,A 0.000,B 0.000,C 90.000,E1 273.555} C_DIS
LIN {X -0.183,Y -492.345,Z 793.517,A 0.000,B 0.000,C 90.000,E1 273.094} C_DIS
LIN {X 0.022,Y -491.806,Z 793.514,A 0.000,B 0.000,C 90.000,E1 272.579} C_DIS
LIN {X 0.229,Y -490.858,Z 793.512,A 0.000,B 0.000,C 90.000,E1 272.064} C_DIS
LIN {X -0.042,Y -489.536,Z 793.509,A 0.000,B 0.000,C 90.000,E1 271.604} C_DIS
LIN {X 0.008,Y -486.684,Z 793.505,A 0.000,B 0.000,C 90.000,E1 270.859} C_DIS
LIN {X 0.190,Y -484.169,Z 793.502,A 0.000,B 0.000,C 90.000,E1 270.344} C_DIS
LIN {X -0.125,Y -481.102,Z 793.499,A 0.000,B 0.000,C 90.000,E1 269.885} C_DIS
LIN {X 0.026,Y -477.301,Z 793.497,A 0.000,B 0.000,C 90.000,E1 269.370} C_DIS
LIN {X 0.154,Y -472.689,Z 793.494,A 0.000,B 0.000,C 90.000,E1 268.854} C_DIS
LIN {X -0.056,Y -467.216,Z 793.491,A 0.000,B 0.000,C 90.000,E1 268.396} C_DIS
LIN {X -0.074,Y -464.129,Z 793.490,A 0.000,B 0.000,C 90.000,E1 268.165} C_DIS
LIN {X -0.157,Y -457.425,Z 793.487,A 0.000,B 0.000,C 90.000,E1 267.764} C_DIS
LIN {X -0.115,Y -450.044,Z 793.486,A 0.000,B 0.000,C 90.000,E1 267.421} C_DIS
LIN {X 0.076,Y -442.458,Z 793.484,A 0.000,B 0.000,C 90.000,E1 267.135} C_DIS
LIN {X -0.145,Y -434.027,Z 793.483,A 0.000,B 0.000,C 90.000,E1 266.963} C_DIS
LIN {X -0.017,Y -426.430,Z 793.482,A 0.000,B 0.000,C 90.000,E1 266.846} C_DIS
LIN {X 0.098,Y -419.927,Z 793.482,A 0.000,B 0.000,C 90.000,E1 266.788} C_DIS
LIN {X 0.017,Y -180.972,Z 793.482,A 0.000,B 0.000,C 90.000,E1 266.788} C_DIS
LIN {X -0.015,Y -180.875,Z 793.473,A 0.000,B 0.000,C 90.000,E1 265.065} C_DIS
LIN {X 0.041,Y -178.991,Z 793.444,A 0.000,B 0.000,C 90.000,E1 259.982} C_DIS
LIN {X 0.052,Y -177.978,Z 793.435,A 0.000,B 0.000,C 90.000,E1 258.285} C_DIS
LIN {X 0.022,Y -175.623,Z 793.411,A 0.000,B 0.000,C 90.000,E1 254.047} C_DIS
LIN {X 0.082,Y -172.343,Z 793.388,A 0.000,B 0.000,C 90.000,E1 249.752} C_DIS
LIN {X 0.061,Y -171.819,Z 793.383,A 0.000,B 0.000,C 90.000,E1 248.901} C_DIS
LIN {X 0.068,Y -170.287,Z 793.373,A 0.000,B 0.000,C 90.000,E1 247.177} C_DIS
LIN {X 0.004,Y -166.826,Z 793.349,A 0.000,B 0.000,C 90.000,E1 242.871} C_DIS
LIN {X -0.079,Y -162.808,Z 793.325,A 0.000,B 0.000,C 90.000,E1 238.535} C_DIS
LIN {X -0.015,Y -161.495,Z 793.315,A 0.000,B 0.000,C 90.000,E1 236.755} C_DIS
LIN {X -0.061,Y -157.492,Z 793.291,A 0.000,B 0.000,C 90.000,E1 232.351} C_DIS
LIN {X -0.027,Y -155.510,Z 793.276,A 0.000,B 0.000,C 90.000,E1 229.666} C_DIS
LIN {X 0.023,Y -151.812,Z 793.251,A 0.000,B 0.000,C 90.000,E1 225.162} C_DIS
LIN {X 0.036,Y -150.024,Z 793.236,A 0.000,B 0.000,C 90.000,E1 222.447} C_DIS
LIN {X -0.050,Y -146.845,Z 793.211,A 0.000,B 0.000,C 90.000,E1 217.935} C_DIS
LIN {X -0.031,Y -145.429,Z 793.195,A 0.000,B 0.000,C 90.000,E1 215.185} C_DIS
LIN {X -0.035,Y -142.852,Z 793.170,A 0.000,B 0.000,C 90.000,E1 210.590} C_DIS
LIN {X 0.017,Y -141.468,Z 793.149,A 0.000,B 0.000,C 90.000,E1 206.873} C_DIS
LIN {X 0.008,Y -139.377,Z 793.113,A 0.000,B 0.000,C 90.000,E1 200.375} C_DIS
LIN {X -0.002,Y -138.829,Z 793.098,A 0.000,B 0.000,C 90.000,E1 197.583} C_DIS
LIN {X -0.074,Y -138.353,Z 793.056,A 0.000,B 0.000,C 90.000,E1 190.141} C_DIS
LIN {X 0.060,Y -139.528,Z 793.004,A 0.000,B 0.000,C 90.000,E1 180.745} C_DIS
LIN {X 0.014,Y -141.202,Z 792.973,A 0.000,B 0.000,C 90.000,E1 175.179} C_DIS
LIN {X -0.027,Y -142.578,Z 792.958,A 0.000,B 0.000,C 90.000,E1 172.413} C_DIS
LIN {X 0.068,Y -144.870,Z 792.932,A 0.000,B 0.000,C 90.000,E1 167.757} C_DIS
LIN {X 0.023,Y -147.498,Z 792.912,A 0.000,B 0.000,C 90.000,E1 164.102} C_DIS
LIN {X -0.043,Y -150.087,Z 792.891,A 0.000,B 0.000,C 90.000,E1 160.477} C_DIS
LIN {X -0.030,Y -153.439,Z 792.871,A 0.000,B 0.000,C 90.000,E1 156.847} C_DIS
LIN {X -0.036,Y -157.803,Z 792.846,A 0.000,B 0.000,C 90.000,E1 152.359} C_DIS
LIN {X -0.004,Y -162.084,Z 792.827,A 0.000,B 0.000,C 90.000,E1 148.791} C_DIS
LIN {X 0.021,Y -166.283,Z 792.807,A 0.000,B 0.000,C 90.000,E1 145.261} C_DIS
LIN {X 0.018,Y -171.300,Z 792.788,A 0.000,B 0.000,C 90.000,E1 141.778} C_DIS
LIN {X 0.054,Y -176.197,Z 792.769,A 0.000,B 0.000,C 90.000,E1 138.324} C_DIS
LIN {X -0.082,Y -180.472,Z 792.754,A 0.000,B 0.000,C 90.000,E1 135.810} C_DIS
LIN {X 0.030,Y -185.876,Z 792.736,A 0.000,B 0.000,C 90.000,E1 132.405} C_DIS
LIN {X -0.054,Y -190.501,Z 792.722,A 0.000,B 0.000,C 90.000,E1 129.930} C_DIS
LIN {X 0.031,Y -192.576,Z 792.715,A 0.000,B 0.000,C 90.000,E1 128.669} C_DIS
LIN {X 0.012,Y -292.717,Z 792.715,A 0.000,B 0.000,C 90.000,E1 128.669} C_DIS
LIN {X 0.035,Y -294.765,Z 792.715,A 0.000,B 0.000,C 90.000,E1 128.624} C_DIS
LIN {X -0.087,Y -298.556,Z 792.714,A 0.000,B 0.000,C 90.000,E1 128.463} C_DIS
LIN {X 0.023,Y -300.812,Z 792.713,A 0.000,B 0.000,C 90.000,E1 128.257} C_DIS
LIN {X -0.158,Y -304.676,Z 792.710,A 0.000,B 0.000,C 90.000,E1 127.810} C_DIS
LIN {X 0.035,Y -306.508,Z 792.708,A 0.000,B 0.000,C 90.000,E1 127.443} C_DIS
LIN {X 0.046,Y -307.937,Z 792.706,A 0.000,B 0.000,C 90.000,E1 127.111} C_DIS
LIN {X 0.043,Y -309.983,Z 792.703,A 0.000,B 0.000,C 90.000,E1 126.457} C_DIS
LIN {X -0.086,Y -320.061,Z 792.685,A 0.000,B 0.000,C 90.000,E1 123.245} C_DIS
LIN {X -0.081,Y -330.451,Z 792.669,A 0.000,B 0.000,C 90.000,E1 120.384} C_DIS
LIN {X -0.009,Y -342.194,Z 792.653,A 0.000,B 0.000,C 90.000,E1 117.564} C_DIS
LIN {X -0.068,Y -355.391,Z 792.638,A 0.000,B 0.000,C 90.000,E1 114.823} C_DIS
LIN {X 0.065,Y -368.438,Z 792.625,A 0.000,B 0.000,C 90.000,E1 112.408} C_DIS
LIN {X 0.062,Y -382.821,Z 792.612,A 0.000,B 0.000,C 90.000,E1 110.066} C_DIS
LIN {X 0.156,Y -398.644,Z 792.599,A 0.000,B 0.000,C 90.000,E1 107.764} C_DIS
LIN {X 0.020,Y -416.020,Z 792.586,A 0.000,B 0.000,C 90.000,E1 105.552} C_DIS
LIN {X 0.208,Y -435.060,Z 792.574,A 0.000,B 0.000,C 90.000,E1 103.355} C_DIS
LIN {X -0.174,Y -455.161,Z 792.563,A 0.000,B 0.000,C 90.000,E1 101.366} C_DIS
LIN {X 0.120,Y -467.970,Z 792.556,A 0.000,B 0.000,C 90.000,E1 100.141} C_DIS
LIN {X 0.126,Y -469.999,Z 792.555,A 0.000,B 0.000,C 90.000,E1 99.905} C_DIS
LIN {X 0.131,Y -471.542,Z 792.554,A 0.000,B 0.000,C 90.000,E1 99.670} C_DIS
LIN {X -0.093,Y -472.805,Z 792.552,A 0.000,B 0.000,C 90.000,E1 99.443} C_DIS
LIN {X -0.238,Y -473.732,Z 792.551,A 0.000,B 0.000,C 90.000,E1 99.208} C_DIS
LIN {X -0.051,Y -474.751,Z 792.548,A 0.000,B 0.000,C 90.000,E1 98.681} C_DIS
LIN {X 0.070,Y -474.784,Z 792.545,A 0.000,B 0.000,C 90.000,E1 98.163} C_DIS
LIN {X 0.199,Y -473.841,Z 792.543,A 0.000,B 0.000,C 90.000,E1 97.644} C_DIS
LIN {X -0.140,Y -471.765,Z 792.540,A 0.000,B 0.000,C 90.000,E1 97.182} C_DIS
LIN {X 0.043,Y -454.021,Z 792.524,A 0.000,B 0.000,C 90.000,E1 94.359} C_DIS
LIN {X -0.064,Y -441.983,Z 792.513,A 0.000,B 0.000,C 90.000,E1 92.293} C_DIS
LIN {X 0.101,Y -432.736,Z 792.504,A 0.000,B 0.000,C 90.000,E1 90.688} C_DIS
LIN {X -0.206,Y -421.640,Z 792.493,A 0.000,B 0.000,C 90.000,E1 88.854} C_DIS
LIN {X 0.101,Y -410.312,Z 792.483,A 0.000,B 0.000,C 90.000,E1 86.906} C_DIS
LIN {X 0.135,Y -400.533,Z 792.474,A 0.000,B 0.000,C 90.000,E1 85.241} C_DIS
LIN {X 0.135,Y -385.918,Z 792.460,A 0.000,B 0.000,C 90.000,E1 82.704} C_DIS
LIN {X -0.143,Y -373.363,Z 792.447,A 0.000,B 0.000,C 90.000,E1 80.443} C_DIS
LIN {X 0.039,Y -356.710,Z 792.429,A 0.000,B 0.000,C 90.000,E1 77.173} C_DIS
LIN {X 0.148,Y -346.510,Z 792.417,A 0.000,B 0.000,C 90.000,E1 75.046} C_DIS
LIN {X 0.120,Y -336.447,Z 792.405,A 0.000,B 0.000,C 90.000,E1 72.906} C_DIS
LIN {X 0.041,Y -325.169,Z 792.391,A 0.000,B 0.000,C 90.000,E1 70.423} C_DIS
LIN {X 0.145,Y -312.774,Z 792.375,A 0.000,B 0.000,C 90.000,E1 67.539} C_DIS
LIN {X 0.030,Y -298.771,Z 792.355,A 0.000,B 0.000,C 90.000,E1 63.973} C_DIS
LIN {X -0.132,Y -287.024,Z 792.337,A 0.000,B 0.000,C 90.000,E1 60.667} C_DIS
LIN {X -0.019,Y -277.114,Z 792.320,A 0.000,B 0.000,C 90.000,E1 57.582} C_DIS
LIN {X -0.022,Y -268.648,Z 792.305,A 0.000,B 0.000,C 90.000,E1 54.815} C_DIS
LIN {X -0.052,Y -262.450,Z 792.293,A 0.000,B 0.000,C 90.000,E1 52.718} C_DIS
LIN {X 0.150,Y -254.197,Z 792.277,A 0.000,B 0.000,C 90.000,E1 49.828} C_DIS
LIN {X -0.069,Y -246.157,Z 792.261,A 0.000,B 0.000,C 90.000,E1 46.986} C_DIS
LIN {X -0.031,Y -236.740,Z 792.240,A 0.000,B 0.000,C 90.000,E1 43.299} C_DIS
LIN {X 0.002,Y -229.538,Z 792.224,A 0.000,B 0.000,C 90.000,E1 40.297} C_DIS
LIN {X 0.087,Y -222.591,Z 792.207,A 0.000,B 0.000,C 90.000,E1 37.237} C_DIS
LIN {X 0.101,Y -214.333,Z 792.186,A 0.000,B 0.000,C 90.000,E1 33.372} C_DIS
LIN {X 0.024,Y -208.349,Z 792.168,A 0.000,B 0.000,C 90.000,E1 30.256} C_DIS
LIN {X 0.031,Y -203.045,Z 792.150,A 0.000,B 0.000,C 90.000,E1 27.078} C_DIS
LIN {X -0.042,Y -197.500,Z 792.128,A 0.000,B 0.000,C 90.000,E1 23.078} C_DIS
LIN {X -0.057,Y -192.991,Z 792.106,A 0.000,B 0.000,C 90.000,E1 19.014} C_DIS
LIN {X -0.026,Y -189.631,Z 792.083,A 0.000,B 0.000,C 90.000,E1 14.898} C_DIS
LIN {X -0.005,Y -186.786,Z 792.051,A 0.000,B 0.000,C 90.000,E1 9.095} C_DIS
LIN {X -0.025,Y -187.891,Z 791.970,A 0.000,B 0.000,C 90.000,E1 354.546} C_DIS
LIN {X 0.004,Y -190.839,Z 791.942,A 0.000,B 0.000,C 90.000,E1 349.567} C_DIS
LIN {X -0.034,Y -194.283,Z 791.919,A 0.000,B 0.000,C 90.000,E1 345.463} C_DIS
LIN {X -0.103,Y -198.652,Z 791.896,A 0.000,B 0.000,C 90.000,E1 341.402} C_DIS
LIN {X -0.093,Y -204.128,Z 791.874,A 0.000,B 0.000,C 90.000,E1 337.358} C_DIS
LIN {X -0.061,Y -209.202,Z 791.856,A 0.000,B 0.000,C 90.000,E1 334.152} C_DIS
LIN {X -0.058,Y -216.386,Z 791.834,A 0.000,B 0.000,C 90.000,E1 330.205} C_DIS
LIN {X -0.044,Y -222.679,Z 791.817,A 0.000,B 0.000,C 90.000,E1 327.089} C_DIS
LIN {X -0.042,Y -231.171,Z 791.796,A 0.000,B 0.000,C 90.000,E1 323.256} C_DIS
LIN {X 0.088,Y -240.407,Z 791.775,A 0.000,B 0.000,C 90.000,E1 319.461} C_DIS
LIN {X 0.108,Y -249.507,Z 791.756,A 0.000,B 0.000,C 90.000,E1 316.134} C_DIS
LIN {X 0.025,Y -259.257,Z 791.738,A 0.000,B 0.000,C 90.000,E1 312.894} C_DIS
LIN {X -0.027,Y -271.058,Z 791.719,A 0.000,B 0.000,C 90.000,E1 309.358} C_DIS
LIN {X 0.010,Y -284.025,Z 791.699,A 0.000,B 0.000,C 90.000,E1 305.884} C_DIS
LIN {X 0.046,Y -295.410,Z 791.684,A 0.000,B 0.000,C 90.000,E1 303.166} C_DIS
LIN {X -0.111,Y -308.023,Z 791.670,A 0.000,B 0.000,C 90.000,E1 300.541} C_DIS
LIN {X 0.096,Y -320.201,Z 791.657,A 0.000,B 0.000,C 90.000,E1 298.231} C_DIS
LIN {X 0.040,Y -338.870,Z 791.639,A 0.000,B 0.000,C 90.000,E1 295.079} C_DIS
LIN {X -0.113,Y -353.104,Z 791.627,A 0.000,B 0.000,C 90.000,E1 292.950} C_DIS
LIN {X -0.145,Y -370.839,Z 791.614,A 0.000,B 0.000,C 90.000,E1 290.556} C_DIS
LIN {X -0.143,Y -392.790,Z 791.600,A 0.000,B 0.000,C 90.000,E1 287.946} C_DIS
LIN {X -0.204,Y -407.941,Z 791.590,A 0.000,B 0.000,C 90.000,E1 286.260} C_DIS
LIN {X 0.166,Y -420.432,Z 791.583,A 0.000,B 0.000,C 90.000,E1 284.828} C_DIS
LIN {X 0.149,Y -432.595,Z 791.575,A 0.000,B 0.000,C 90.000,E1 283.480} C_DIS
LIN {X -0.062,Y -444.454,Z 791.568,A 0.000,B 0.000,C 90.000,E1 282.175} C_DIS
LIN {X -0.104,Y -453.367,Z 791.562,A 0.000,B 0.000,C 90.000,E1 281.130} C_DIS
LIN {X 0.049,Y -461.627,Z 791.556,A 0.000,B 0.000,C 90.000,E1 280.074} C_DIS
LIN {X 0.219,Y -469.257,Z 791.550,A 0.000,B 0.000,C 90.000,E1 279.029} C_DIS
LIN {X 0.157,Y -474.555,Z 791.546,A 0.000,B 0.000,C 90.000,E1 278.276} C_DIS
LIN {X 0.072,Y -479.348,Z 791.542,A 0.000,B 0.000,C 90.000,E1 277.530} C_DIS
LIN {X 0.099,Y -483.510,Z 791.538,A 0.000,B 0.000,C 90.000,E1 276.777} C_DIS
LIN {X 0.102,Y -486.884,Z 791.534,A 0.000,B 0.000,C 90.000,E1 276.030} C_DIS
LIN {X -0.183,Y -488.753,Z 791.531,A 0.000,B 0.000,C 90.000,E1 275.568} C_DIS
LIN {X 0.022,Y -490.236,Z 791.528,A 0.000,B 0.000,C 90.000,E1 275.049} C_DIS
LIN {X 0.237,Y -491.384,Z 791.525,A 0.000,B 0.000,C 90.000,E1 274.531} C_DIS
LIN {X -0.067,Y -492.131,Z 791.523,A 0.000,B 0.000,C 90.000,E1 274.073} C_DIS
LIN {X 0.162,Y -492.433,Z 791.520,A 0.000,B 0.000,C 90.000,E1 273.555} C_DIS
LIN {X -0.100,Y -492.349,Z 791.517,A 0.000,B 0.000,C 90.000,E1 273.094} C_DIS
LIN {X 0.104,Y -491.858,Z 791.514,A 0.000,B 0.000,C 90.000,E1 272.579} C_DIS
LIN {X -0.180,Y -490.955,Z 791.512,A 0.000,B 0.000,C 90.000,E1 272.121} C_DIS
LIN {X 0.041,Y -489.632,Z 791.509,A 0.000,B 0.000,C 90.000,E1 271.604} C_DIS
LIN {X 0.238,Y -487.879,Z 791.506,A 0.000,B 0.000,C 90.000,E1 271.088} C_DIS
LIN {X -0.057,Y -485.674,Z 791.503,A 0.000,B 0.000,C 90.000,E1 270.630} C_DIS
LIN {X 0.119,Y -482.909,Z 791.501,A 0.000,B 0.000,C 90.000,E1 270.115} C_DIS
LIN {X -0.201,Y -479.477,Z 791.498,A 0.000,B 0.000,C 90.000,E1 269.656} C_DIS
LIN {X 0.109,Y -477.571,Z 791.497,A 0.000,B 0.000,C 90.000,E1 269.370} C_DIS
LIN {X -0.235,Y -472.947,Z 791.494,A 0.000,B 0.000,C 90.000,E1 268.912} C_DIS
LIN {X -0.012,Y -467.510,Z 791.491,A 0.000,B 0.000,C 90.000,E1 268.396} C_DIS
LIN {X 0.129,Y -461.274,Z 791.489,A 0.000,B 0.000,C 90.000,E1 267.936} C_DIS
LIN {X -0.136,Y -457.766,Z 791.487,A 0.000,B 0.000,C 90.000,E1 267.764} C_DIS
LIN {X -0.094,Y -450.440,Z 791.486,A 0.000,B 0.000,C 90.000,E1 267.421} C_DIS
LIN {X 0.082,Y -443.035,Z 791.484,A 0.000,B 0.000,C 90.000,E1 267.135} C_DIS
LIN {X -0.211,Y -434.395,Z 791.483,A 0.000,B 0.000,C 90.000,E1 266.963} C_DIS
LIN {X -0.109,Y -426.919,Z 791.482,A 0.000,B 0.000,C 90.000,E1 266.846} C_DIS
LIN {X -0.001,Y -419.862,Z 791.482,A 0.000,B 0.000,C 90.000,E1 266.788} C_DIS
LIN {X -0.025,Y -180.971,Z 791.482,A 0.000,B 0.000,C 90.000,E1 266.788} C_DIS
LIN {X -0.055,Y -180.872,Z 791.472,A 0.000,B 0.000,C 90.000,E1 265.065} C_DIS
LIN {X 0.002,Y -178.989,Z 791.444,A 0.000,B 0.000,C 90.000,E1 259.982} C_DIS
LIN {X 0.014,Y -177.970,Z 791.435,A 0.000,B 0.000,C 90.000,E1 258.285} C_DIS
LIN {X 0.032,Y -175.613,Z 791.411,A 0.000,B 0.000,C 90.000,E1 254.031} C_DIS
LIN {X 0.044,Y -172.335,Z 791.388,A 0.000,B 0.000,C 90.000,E1 249.752} C_DIS
LIN {X 0.023,Y -171.812,Z 791.383,A 0.000,B 0.000,C 90.000,E1 248.901} C_DIS
LIN {X 0.031,Y -170.276,Z 791.373,A 0.000,B 0.000,C 90.000,E1 247.177} C_DIS
LIN {X -0.034,Y -166.817,Z 791.349,A 0.000,B 0.000,C 90.000,E1 242.871} C_DIS
LIN {X 0.023,Y -162.798,Z 791.325,A 0.000,B 0.000,C 90.000,E1 238.486} C_DIS
LIN {X -0.051,Y -161.485,Z 791.315,A 0.000,B 0.000,C 90.000,E1 236.755} C_DIS
LIN {X -0.001,Y -157.482,Z 791.291,A 0.000,B 0.000,C 90.000,E1 232.316} C_DIS
LIN {X 0.057,Y -155.498,Z 791.276,A 0.000,B 0.000,C 90.000,E1 229.622} C_DIS
LIN {X -0.012,Y -151.803,Z 791.251,A 0.000,B 0.000,C 90.000,E1 225.162} C_DIS
LIN {X 0.001,Y -150.013,Z 791.236,A 0.000,B 0.000,C 90.000,E1 222.447} C_DIS
LIN {X 0.032,Y -146.837,Z 791.211,A 0.000,B 0.000,C 90.000,E1 217.890} C_DIS
LIN {X 0.018,Y -145.419,Z 791.195,A 0.000,B 0.000,C 90.000,E1 215.152} C_DIS
LIN {X 0.054,Y -142.847,Z 791.170,A 0.000,B 0.000,C 90.000,E1 210.541} C_DIS
LIN {X -0.016,Y -141.461,Z 791.149,A 0.000,B 0.000,C 90.000,E1 206.873} C_DIS
LIN {X -0.026,Y -139.375,Z 791.113,A 0.000,B 0.000,C 90.000,E1 200.375} C_DIS
LIN {X -0.035,Y -138.825,Z 791.098,A 0.000,B 0.000,C 90.000,E1 197.583} C_DIS
LIN {X 0.053,Y -138.353,Z 791.056,A 0.000,B 0.000,C 90.000,E1 190.074} C_DIS
LIN {X 0.027,Y -139.530,Z 791.004,A 0.000,B 0.000,C 90.000,E1 180.745} C_DIS
LIN {X -0.020,Y -141.208,Z 790.973,A 0.000,B 0.000,C 90.000,E1 175.179} C_DIS
LIN {X -0.062,Y -142.583,Z 790.958,A 0.000,B 0.000,C 90.000,E1 172.413} C_DIS
LIN {X 0.034,Y -144.879,Z 790.932,A 0.000,B 0.000,C 90.000,E1 167.757} C_DIS
LIN {X -0.012,Y -147.506,Z 790.912,A 0.000,B 0.000,C 90.000,E1 164.102} C_DIS
LIN {X 0.063,Y -150.099,Z 790.891,A 0.000,B 0.000,C 90.000,E1 160.423} C_DIS
LIN {X 0.075,Y -153.454,Z 790.871,A 0.000,B 0.000,C 90.000,E1 156.794} C_DIS
LIN {X -0.073,Y -157.817,Z 790.846,A 0.000,B 0.000,C 90.000,E1 152.359} C_DIS
LIN {X -0.041,Y -162.100,Z 790.827,A 0.000,B 0.000,C 90.000,E1 148.791} C_DIS
LIN {X -0.017,Y -166.300,Z 790.807,A 0.000,B 0.000,C 90.000,E1 145.261} C_DIS
LIN {X -0.019,Y -171.317,Z 790.788,A 0.000,B 0.000,C 90.000,E1 141.778} C_DIS
LIN {X 0.015,Y -176.216,Z 790.768,A 0.000,B 0.000,C 90.000,E1 138.324} C_DIS
LIN {X 0.009,Y -180.494,Z 790.754,A 0.000,B 0.000,C 90.000,E1 135.769} C_DIS
LIN {X -0.010,Y -185.897,Z 790.736,A 0.000,B 0.000,C 90.000,E1 132.405} C_DIS
LIN {X 0.051,Y -190.524,Z 790.722,A 0.000,B 0.000,C 90.000,E1 129.886} C_DIS
LIN {X 0.070,Y -192.556,Z 790.715,A 0.000,B 0.000,C 90.000,E1 128.669} C_DIS
LIN {X 0.064,Y -292.293,Z 790.715,A 0.000,B 0.000,C 90.000,E1 128.669} C_DIS
LIN {X 0.020,Y -293.123,Z 790.715,A 0.000,B 0.000,C 90.000,E1 128.669} C_DIS
LIN {X -0.010,Y -298.399,Z 790.714,A 0.000,B 0.000,C 90.000,E1 128.463} C_DIS
LIN {X -0.040,Y -300.970,Z 790.713,A 0.000,B 0.000,C 90.000,E1 128.257} C_DIS
LIN {X 0.191,Y -304.773,Z 790.710,A 0.000,B 0.000,C 90.000,E1 127.729} C_DIS
LIN {X -0.042,Y -306.572,Z 790.708,A 0.000,B 0.000,C 90.000,E1 127.443} C_DIS
LIN {X 0.153,Y -307.979,Z 790.706,A 0.000,B 0.000,C 90.000,E1 127.076} C_DIS
LIN {X -0.035,Y -310.004,Z 790.703,A 0.000,B 0.000,C 90.000,E1 126.457} C_DIS
LIN {X 0.010,Y -320.089,Z 790.685,A 0.000,B 0.000,C 90.000,E1 123.214} C_DIS
LIN {X 0.122,Y -330.485,Z 790.669,A 0.000,B 0.000,C 90.000,E1 120.335} C_DIS
LIN {X 0.211,Y -342.235,Z 790.653,A 0.000,B 0.000,C 90.000,E1 117.513} C_DIS
LIN {X 0.169,Y -355.438,Z 790.638,A 0.000,B 0.000,C 90.000,E1 114.771} C_DIS
LIN {X 0.118,Y -368.493,Z 790.624,A 0.000,B 0.000,C 90.000,E1 112.386} C_DIS
LIN {X -0.027,Y -382.884,Z 790.611,A 0.000,B 0.000,C 90.000,E1 110.066} C_DIS
LIN {X 0.065,Y -398.716,Z 790.599,A 0.000,B 0.000,C 90.000,E1 107.764} C_DIS
LIN {X -0.074,Y -416.101,Z 790.586,A 0.000,B 0.000,C 90.000,E1 105.552} C_DIS
LIN {X 0.113,Y -435.149,Z 790.574,A 0.000,B 0.000,C 90.000,E1 103.355} C_DIS
LIN {X -0.177,Y -455.254,Z 790.563,A 0.000,B 0.000,C 90.000,E1 101.355} C_DIS
LIN {X 0.029,Y -468.055,Z 790.556,A 0.000,B 0.000,C 90.000,E1 100.141} C_DIS
LIN {X 0.031,Y -470.068,Z 790.555,A 0.000,B 0.000,C 90.000,E1 99.905} C_DIS
LIN {X 0.031,Y -471.600,Z 790.554,A 0.000,B 0.000,C 90.000,E1 99.670} C_DIS
LIN {X -0.115,Y -472.850,Z 790.552,A 0.000,B 0.000,C 90.000,E1 99.434} C_DIS
LIN {X 0.129,Y -473.767,Z 790.551,A 0.000,B 0.000,C 90.000,E1 99.151} C_DIS
LIN {X -0.151,Y -474.767,Z 790.548,A 0.000,B 0.000,C 90.000,E1 98.681} C_DIS
LIN {X -0.030,Y -474.784,Z 790.545,A 0.000,B 0.000,C 90.000,E1 98.163} C_DIS
LIN {X 0.100,Y -473.824,Z 790.543,A 0.000,B 0.000,C 90.000,E1 97.644} C_DIS
LIN {X -0.239,Y -471.724,Z 790.540,A 0.000,B 0.000,C 90.000,E1 97.182} C_DIS
LIN {X -0.053,Y -453.979,Z 790.524,A 0.000,B 0.000,C 90.000,E1 94.359} C_DIS
LIN {X -0.159,Y -441.934,Z 790.513,A 0.000,B 0.000,C 90.000,E1 92.293} C_DIS
LIN {X 0.008,Y -432.704,Z 790.504,A 0.000,B 0.000,C 90.000,E1 90.688} C_DIS
LIN {X 0.124,Y -421.586,Z 790.493,A 0.000,B 0.000,C 90.000,E1 88.797} C_DIS
LIN {X 0.011,Y -410.274,Z 790.483,A 0.000,B 0.000,C 90.000,E1 86.906} C_DIS
LIN {X 0.046,Y -400.519,Z 790.474,A 0.000,B 0.000,C 90.000,E1 85.241} C_DIS
LIN {X 0.049,Y -385.903,Z 790.460,A 0.000,B 0.000,C 90.000,E1 82.704} C_DIS
LIN {X 0.142,Y -373.364,Z 790.447,A 0.000,B 0.000,C 90.000,E1 80.387} C_DIS
LIN {X -0.081,Y -355.291,Z 790.427,A 0.000,B 0.000,C 90.000,E1 76.881} C_DIS
LIN {X -0.006,Y -345.102,Z 790.415,A 0.000,B 0.000,C 90.000,E1 74.755} C_DIS
LIN {X -0.077,Y -333.652,Z 790.402,A 0.000,B 0.000,C 90.000,E1 72.308} C_DIS
LIN {X 0.194,Y -322.452,Z 790.388,A 0.000,B 0.000,C 90.000,E1 69.752} C_DIS
LIN {X 0.164,Y -307.637,Z 790.368,A 0.000,B 0.000,C 90.000,E1 66.230} C_DIS
LIN {X 0.135,Y -294.099,Z 790.348,A 0.000,B 0.000,C 90.000,E1 62.615} C_DIS
LIN {X 0.000,Y -283.838,Z 790.331,A 0.000,B 0.000,C 90.000,E1 59.616} C_DIS
LIN {X -0.156,Y -275.212,Z 790.316,A 0.000,B 0.000,C 90.000,E1 56.914} C_DIS
LIN {X -0.053,Y -266.870,Z 790.301,A 0.000,B 0.000,C 90.000,E1 54.116} C_DIS
LIN {X 0.040,Y -260.711,Z 790.289,A 0.000,B 0.000,C 90.000,E1 51.984} C_DIS
LIN {X 0.003,Y -252.507,Z 790.273,A 0.000,B 0.000,C 90.000,E1 49.138} C_DIS
LIN {X 0.080,Y -242.701,Z 790.253,A 0.000,B 0.000,C 90.000,E1 45.486} C_DIS
LIN {X 0.079,Y -235.282,Z 790.236,A 0.000,B 0.000,C 90.000,E1 42.528} C_DIS
LIN {X -0.075,Y -228.136,Z 790.220,A 0.000,B 0.000,C 90.000,E1 39.564} C_DIS
LIN {X -0.021,Y -221.231,Z 790.203,A 0.000,B 0.000,C 90.000,E1 36.503} C_DIS
LIN {X -0.051,Y -214.668,Z 790.186,A 0.000,B 0.000,C 90.000,E1 33.420} C_DIS
LIN {X 0.058,Y -208.692,Z 790.168,A 0.000,B 0.000,C 90.000,E1 30.256} C_DIS
LIN {X -0.108,Y -203.359,Z 790.151,A 0.000,B 0.000,C 90.000,E1 27.129} C_DIS
LIN {X 0.008,Y -197.791,Z 790.128,A 0.000,B 0.000,C 90.000,E1 23.078} C_DIS
LIN {X -0.063,Y -193.290,Z 790.106,A 0.000,B 0.000,C 90.000,E1 19.033} C_DIS
LIN {X 0.038,Y -189.905,Z 790.083,A 0.000,B 0.000,C 90.000,E1 14.898} C_DIS
LIN {X 0.070,Y -187.016,Z 790.051,A 0.000,B 0.000,C 90.000,E1 9.095} C_DIS
LIN {X -0.018,Y -188.056,Z 789.970,A 0.000,B 0.000,C 90.000,E1 354.546} C_DIS
LIN {X 0.017,Y -190.996,Z 789.942,A 0.000,B 0.000,C 90.000,E1 349.567} C_DIS
LIN {X -0.015,Y -194.425,Z 789.919,A 0.000,B 0.000,C 90.000,E1 345.463} C_DIS
LIN {X -0.081,Y -198.800,Z 789.897,A 0.000,B 0.000,C 90.000,E1 341.402} C_DIS
LIN {X -0.065,Y -204.281,Z 789.874,A 0.000,B 0.000,C 90.000,E1 337.358} C_DIS
LIN {X 0.068,Y -210.706,Z 789.852,A 0.000,B 0.000,C 90.000,E1 333.332} C_DIS
LIN {X 0.035,Y -218.078,Z 789.830,A 0.000,B 0.000,C 90.000,E1 329.410} C_DIS
LIN {X 0.005,Y -226.110,Z 789.809,A 0.000,B 0.000,C 90.000,E1 325.548} C_DIS
LIN {X 0.006,Y -234.891,Z 789.787,A 0.000,B 0.000,C 90.000,E1 321.743} C_DIS
LIN {X 0.039,Y -244.443,Z 789.767,A 0.000,B 0.000,C 90.000,E1 318.000} C_DIS
LIN {X 0.006,Y -254.880,Z 789.746,A 0.000,B 0.000,C 90.000,E1 314.352} C_DIS
LIN {X -0.088,Y -265.075,Z 789.729,A 0.000,B 0.000,C 90.000,E1 311.148} C_DIS
LIN {X -0.008,Y -276.094,Z 789.711,A 0.000,B 0.000,C 90.000,E1 307.971} C_DIS
LIN {X 0.021,Y -289.544,Z 789.692,A 0.000,B 0.000,C 90.000,E1 304.532} C_DIS
LIN {X -0.138,Y -299.926,Z 789.679,A 0.000,B 0.000,C 90.000,E1 302.212} C_DIS
LIN {X 0.128,Y -314.765,Z 789.662,A 0.000,B 0.000,C 90.000,E1 299.205} C_DIS
LIN {X -0.008,Y -329.245,Z 789.648,A 0.000,B 0.000,C 90.000,E1 296.668} C_DIS
LIN {X -0.087,Y -346.751,Z 789.633,A 0.000,B 0.000,C 90.000,E1 293.875} C_DIS
LIN {X -0.094,Y -366.061,Z 789.617,A 0.000,B 0.000,C 90.000,E1 291.153} C_DIS
LIN {X -0.163,Y -380.162,Z 789.608,A 0.000,B 0.000,C 90.000,E1 289.396} C_DIS
LIN {X -0.212,Y -397.527,Z 789.596,A 0.000,B 0.000,C 90.000,E1 287.402} C_DIS
LIN {X -0.019,Y -412.464,Z 789.587,A 0.000,B 0.000,C 90.000,E1 285.717} C_DIS
LIN {X 0.085,Y -427.242,Z 789.578,A 0.000,B 0.000,C 90.000,E1 284.064} C_DIS
LIN {X 0.161,Y -439.191,Z 789.571,A 0.000,B 0.000,C 90.000,E1 282.715} C_DIS
LIN {X 0.158,Y -448.412,Z 789.565,A 0.000,B 0.000,C 90.000,E1 281.658} C_DIS
LIN {X -0.188,Y -457.026,Z 789.559,A 0.000,B 0.000,C 90.000,E1 280.658} C_DIS
LIN {X -0.078,Y -464.993,Z 789.553,A 0.000,B 0.000,C 90.000,E1 279.613} C_DIS
LIN {X 0.133,Y -472.351,Z 789.548,A 0.000,B 0.000,C 90.000,E1 278.568} C_DIS
LIN {X -0.107,Y -478.928,Z 789.542,A 0.000,B 0.000,C 90.000,E1 277.587} C_DIS
LIN {X -0.087,Y -483.155,Z 789.538,A 0.000,B 0.000,C 90.000,E1 276.834} C_DIS
LIN {X 0.087,Y -485.579,Z 789.535,A 0.000,B 0.000,C 90.000,E1 276.315} C_DIS
LIN {X 0.110,Y -488.510,Z 789.531,A 0.000,B 0.000,C 90.000,E1 275.568} C_DIS
LIN {X -0.175,Y -490.086,Z 789.528,A 0.000,B 0.000,C 90.000,E1 275.106} C_DIS
LIN {X 0.038,Y -491.264,Z 789.526,A 0.000,B 0.000,C 90.000,E1 274.588} C_DIS
LIN {X 0.224,Y -492.057,Z 789.523,A 0.000,B 0.000,C 90.000,E1 274.073} C_DIS
LIN {X -0.039,Y -492.423,Z 789.520,A 0.000,B 0.000,C 90.000,E1 273.612} C_DIS
LIN {X 0.190,Y -492.398,Z 789.517,A 0.000,B 0.000,C 90.000,E1 273.094} C_DIS
LIN {X -0.098,Y -491.939,Z 789.515,A 0.000,B 0.000,C 90.000,E1 272.636} C_DIS
LIN {X 0.110,Y -491.095,Z 789.512,A 0.000,B 0.000,C 90.000,E1 272.121} C_DIS
LIN {X -0.160,Y -489.831,Z 789.509,A 0.000,B 0.000,C 90.000,E1 271.661} C_DIS
LIN {X 0.040,Y -488.120,Z 789.506,A 0.000,B 0.000,C 90.000,E1 271.146} C_DIS
LIN {X 0.231,Y -485.929,Z 789.504,A 0.000,B 0.000,C 90.000,E1 270.630} C_DIS
LIN {X -0.076,Y -483.253,Z 789.501,A 0.000,B 0.000,C 90.000,E1 270.172} C_DIS
LIN {X 0.086,Y -479.909,Z 789.498,A 0.000,B 0.000,C 90.000,E1 269.656} C_DIS
LIN {X 0.229,Y -475.850,Z 789.495,A 0.000,B 0.000,C 90.000,E1 269.141} C_DIS
LIN {X -0.124,Y -470.869,Z 789.493,A 0.000,B 0.000,C 90.000,E1 268.682} C_DIS
LIN {X -0.208,Y -468.123,Z 789.491,A 0.000,B 0.000,C 90.000,E1 268.453} C_DIS
LIN {X -0.088,Y -462.009,Z 789.489,A 0.000,B 0.000,C 90.000,E1 267.993} C_DIS
LIN {X 0.098,Y -458.589,Z 789.488,A 0.000,B 0.000,C 90.000,E1 267.764} C_DIS
LIN {X 0.071,Y -451.282,Z 789.486,A 0.000,B 0.000,C 90.000,E1 267.421} C_DIS
LIN {X 0.187,Y -443.821,Z 789.484,A 0.000,B 0.000,C 90.000,E1 267.135} C_DIS
LIN {X -0.179,Y -440.362,Z 789.484,A 0.000,B 0.000,C 90.000,E1 267.078} C_DIS
LIN {X -0.215,Y -431.938,Z 789.483,A 0.000,B 0.000,C 90.000,E1 266.906} C_DIS
LIN {X -0.030,Y -422.829,Z 789.482,A 0.000,B 0.000,C 90.000,E1 266.788} C_DIS
LIN {X -0.107,Y -420.176,Z 789.482,A 0.000,B 0.000,C 90.000,E1 266.788} C_DIS
LIN {X -0.079,Y -180.970,Z 789.482,A 0.000,B 0.000,C 90.000,E1 266.788} C_DIS
LIN {X 0.087,Y -180.869,Z 789.472,A 0.000,B 0.000,C 90.000,E1 265.008} C_DIS
LIN {X -0.036,Y -178.985,Z 789.444,A 0.000,B 0.000,C 90.000,E1 259.982} C_DIS
LIN {X -0.024,Y -177.962,Z 789.435,A 0.000,B 0.000,C 90.000,E1 258.285} C_DIS
LIN {X -0.005,Y -175.605,Z 789.411,A 0.000,B 0.000,C 90.000,E1 254.031} C_DIS
LIN {X 0.007,Y -172.327,Z 789.388,A 0.000,B 0.000,C 90.000,E1 249.752} C_DIS
LIN {X -0.014,Y -171.805,Z 789.383,A 0.000,B 0.000,C 90.000,E1 248.901} C_DIS
LIN {X -0.007,Y -170.264,Z 789.373,A 0.000,B 0.000,C 90.000,E1 247.177} C_DIS
LIN {X -0.070,Y -166.807,Z 789.349,A 0.000,B 0.000,C 90.000,E1 242.871} C_DIS
LIN {X 0.073,Y -162.788,Z 789.325,A 0.000,B 0.000,C 90.000,E1 238.456} C_DIS
LIN {X 0.048,Y -161.477,Z 789.315,A 0.000,B 0.000,C 90.000,E1 236.707} C_DIS
LIN {X -0.036,Y -157.471,Z 789.291,A 0.000,B 0.000,C 90.000,E1 232.316} C_DIS
LIN {X 0.022,Y -155.486,Z 789.276,A 0.000,B 0.000,C 90.000,E1 229.622} C_DIS
LIN {X -0.046,Y -151.794,Z 789.251,A 0.000,B 0.000,C 90.000,E1 225.162} C_DIS
LIN {X -0.033,Y -150.003,Z 789.236,A 0.000,B 0.000,C 90.000,E1 222.447} C_DIS
LIN {X -0.002,Y -146.830,Z 789.211,A 0.000,B 0.000,C 90.000,E1 217.890} C_DIS
LIN {X -0.015,Y -145.411,Z 789.195,A 0.000,B 0.000,C 90.000,E1 215.152} C_DIS
LIN {X 0.021,Y -142.840,Z 789.170,A 0.000,B 0.000,C 90.000,E1 210.541} C_DIS
LIN {X -0.049,Y -141.455,Z 789.149,A 0.000,B 0.000,C 90.000,E1 206.873} C_DIS
LIN {X -0.009,Y -139.373,Z 789.113,A 0.000,B 0.000,C 90.000,E1 200.355} C_DIS
LIN {X -0.068,Y -138.822,Z 789.098,A 0.000,B 0.000,C 90.000,E1 197.583} C_DIS
LIN {X 0.021,Y -138.353,Z 789.056,A 0.000,B 0.000,C 90.000,E1 190.074} C_DIS
LIN {X -0.006,Y -139.533,Z 789.004,A 0.000,B 0.000,C 90.000,E1 180.745} C_DIS
LIN {X -0.053,Y -141.214,Z 788.973,A 0.000,B 0.000,C 90.000,E1 175.179} C_DIS
LIN {X 0.047,Y -142.588,Z 788.958,A 0.000,B 0.000,C 90.000,E1 172.356} C_DIS
LIN {X 0.001,Y -144.887,Z 788.932,A 0.000,B 0.000,C 90.000,E1 167.757} C_DIS
LIN {X -0.045,Y -147.515,Z 788.912,A 0.000,B 0.000,C 90.000,E1 164.102} C_DIS
LIN {X 0.028,Y -150.109,Z 788.891,A 0.000,B 0.000,C 90.000,E1 160.423} C_DIS
LIN {X 0.041,Y -153.468,Z 788.871,A 0.000,B 0.000,C 90.000,E1 156.794} C_DIS
LIN {X 0.032,Y -157.831,Z 788.846,A 0.000,B 0.000,C 90.000,E1 152.308} C_DIS
LIN {X 0.063,Y -162.115,Z 788.826,A 0.000,B 0.000,C 90.000,E1 148.742} C_DIS
LIN {X -0.053,Y -166.316,Z 788.807,A 0.000,B 0.000,C 90.000,E1 145.261} C_DIS
LIN {X 0.049,Y -171.334,Z 788.788,A 0.000,B 0.000,C 90.000,E1 141.743} C_DIS
LIN {X -0.023,Y -176.235,Z 788.768,A 0.000,B 0.000,C 90.000,E1 138.324} C_DIS
LIN {X 0.096,Y -180.515,Z 788.754,A 0.000,B 0.000,C 90.000,E1 135.729} C_DIS
LIN {X 0.077,Y -185.919,Z 788.735,A 0.000,B 0.000,C 90.000,E1 132.366} C_DIS
LIN {X 0.011,Y -190.547,Z 788.722,A 0.000,B 0.000,C 90.000,E1 129.886} C_DIS
LIN {X -0.033,Y -192.547,Z 788.715,A 0.000,B 0.000,C 90.000,E1 128.705} C_DIS
LIN {X 0.090,Y -292.457,Z 788.715,A 0.000,B 0.000,C 90.000,E1 128.669} C_DIS
LIN {X -0.038,Y -294.056,Z 788.715,A 0.000,B 0.000,C 90.000,E1 128.669} C_DIS
LIN {X -0.071,Y -298.628,Z 788.714,A 0.000,B 0.000,C 90.000,E1 128.463} C_DIS
LIN {X -0.102,Y -301.116,Z 788.712,A 0.000,B 0.000,C 90.000,E1 128.257} C_DIS
LIN {X 0.057,Y -304.928,Z 788.710,A 0.000,B 0.000,C 90.000,E1 127.729} C_DIS
LIN {X -0.177,Y -306.684,Z 788.708,A 0.000,B 0.000,C 90.000,E1 127.443} C_DIS
LIN {X 0.018,Y -308.057,Z 788.706,A 0.000,B 0.000,C 90.000,E1 127.076} C_DIS
LIN {X -0.050,Y -315.939,Z 788.692,A 0.000,B 0.000,C 90.000,E1 124.485} C_DIS
LIN {X 0.109,Y -326.949,Z 788.674,A 0.000,B 0.000,C 90.000,E1 121.258} C_DIS
LIN {X 0.097,Y -338.247,Z 788.658,A 0.000,B 0.000,C 90.000,E1 118.437} C_DIS
LIN {X 0.095,Y -350.969,Z 788.643,A 0.000,B 0.000,C 90.000,E1 115.668} C_DIS
LIN {X 0.082,Y -363.559,Z 788.629,A 0.000,B 0.000,C 90.000,E1 113.259} C_DIS
LIN {X -0.053,Y -377.452,Z 788.616,A 0.000,B 0.000,C 90.000,E1 110.918} C_DIS
LIN {X 0.023,Y -392.746,Z 788.603,A 0.000,B 0.000,C 90.000,E1 108.598} C_DIS
LIN {X 0.237,Y -409.551,Z 788.591,A 0.000,B 0.000,C 90.000,E1 106.315} C_DIS
LIN {X -0.164,Y -427.988,Z 788.579,A 0.000,B 0.000,C 90.000,E1 104.175} C_DIS
LIN {X -0.071,Y -447.843,Z 788.567,A 0.000,B 0.000,C 90.000,E1 102.063} C_DIS
LIN {X -0.130,Y -468.220,Z 788.556,A 0.000,B 0.000,C 90.000,E1 100.141} C_DIS
LIN {X -0.139,Y -470.203,Z 788.555,A 0.000,B 0.000,C 90.000,E1 99.905} C_DIS
LIN {X -0.148,Y -471.712,Z 788.554,A 0.000,B 0.000,C 90.000,E1 99.670} C_DIS
LIN {X 0.172,Y -472.935,Z 788.552,A 0.000,B 0.000,C 90.000,E1 99.378} C_DIS
LIN {X -0.050,Y -473.830,Z 788.551,A 0.000,B 0.000,C 90.000,E1 99.151} C_DIS
LIN {X 0.139,Y -474.793,Z 788.548,A 0.000,B 0.000,C 90.000,E1 98.624} C_DIS
LIN {X -0.208,Y -474.775,Z 788.545,A 0.000,B 0.000,C 90.000,E1 98.163} C_DIS
LIN {X -0.079,Y -473.777,Z 788.542,A 0.000,B 0.000,C 90.000,E1 97.644} C_DIS
LIN {X 0.052,Y -471.631,Z 788.540,A 0.000,B 0.000,C 90.000,E1 97.125} C_DIS
LIN {X -0.227,Y -453.879,Z 788.524,A 0.000,B 0.000,C 90.000,E1 94.359} C_DIS
LIN {X 0.112,Y -441.830,Z 788.513,A 0.000,B 0.000,C 90.000,E1 92.236} C_DIS
LIN {X -0.162,Y -432.610,Z 788.504,A 0.000,B 0.000,C 90.000,E1 90.688} C_DIS
LIN {X -0.044,Y -421.492,Z 788.493,A 0.000,B 0.000,C 90.000,E1 88.797} C_DIS
LIN {X -0.154,Y -410.186,Z 788.483,A 0.000,B 0.000,C 90.000,E1 86.906} C_DIS
LIN {X -0.116,Y -400.436,Z 788.473,A 0.000,B 0.000,C 90.000,E1 85.241} C_DIS
LIN {X -0.110,Y -385.826,Z 788.459,A 0.000,B 0.000,C 90.000,E1 82.704} C_DIS
LIN {X -0.013,Y -373.297,Z 788.447,A 0.000,B 0.000,C 90.000,E1 80.387} C_DIS
LIN {X 0.116,Y -355.265,Z 788.427,A 0.000,B 0.000,C 90.000,E1 76.825} C_DIS
LIN {X -0.152,Y -345.092,Z 788.415,A 0.000,B 0.000,C 90.000,E1 74.755} C_DIS
LIN {X 0.100,Y -333.654,Z 788.401,A 0.000,B 0.000,C 90.000,E1 72.253} C_DIS
LIN {X 0.013,Y -321.094,Z 788.386,A 0.000,B 0.000,C 90.000,E1 69.444} C_DIS
LIN {X -0.057,Y -306.425,Z 788.366,A 0.000,B 0.000,C 90.000,E1 65.921} C_DIS
LIN {X 0.017,Y -293.040,Z 788.346,A 0.000,B 0.000,C 90.000,E1 62.281} C_DIS
LIN {X 0.031,Y -284.008,Z 788.331,A 0.000,B 0.000,C 90.000,E1 59.587} C_DIS
LIN {X 0.119,Y -275.432,Z 788.316,A 0.000,B 0.000,C 90.000,E1 56.834} C_DIS
LIN {X 0.067,Y -267.137,Z 788.300,A 0.000,B 0.000,C 90.000,E1 54.069} C_DIS
LIN {X -0.049,Y -260.999,Z 788.289,A 0.000,B 0.000,C 90.000,E1 51.984} C_DIS
LIN {X -0.076,Y -252.837,Z 788.273,A 0.000,B 0.000,C 90.000,E1 49.138} C_DIS
LIN {X 0.014,Y -243.042,Z 788.253,A 0.000,B 0.000,C 90.000,E1 45.486} C_DIS
LIN {X 0.023,Y -235.631,Z 788.236,A 0.000,B 0.000,C 90.000,E1 42.528} C_DIS
LIN {X -0.121,Y -228.451,Z 788.220,A 0.000,B 0.000,C 90.000,E1 39.564} C_DIS
LIN {X -0.058,Y -221.544,Z 788.203,A 0.000,B 0.000,C 90.000,E1 36.503} C_DIS
LIN {X -0.019,Y -213.418,Z 788.181,A 0.000,B 0.000,C 90.000,E1 32.625} C_DIS
LIN {X 0.061,Y -207.595,Z 788.164,A 0.000,B 0.000,C 90.000,E1 29.461} C_DIS
LIN {X 0.046,Y -202.442,Z 788.146,A 0.000,B 0.000,C 90.000,E1 26.283} C_DIS
LIN {X -0.034,Y -197.072,Z 788.124,A 0.000,B 0.000,C 90.000,E1 22.280} C_DIS
LIN {X 0.059,Y -192.794,Z 788.101,A 0.000,B 0.000,C 90.000,E1 18.181} C_DIS
LIN {X 0.067,Y -189.095,Z 788.074,A 0.000,B 0.000,C 90.000,E1 13.244} C_DIS
LIN {X 0.081,Y -186.586,Z 788.037,A 0.000,B 0.000,C 90.000,E1 6.606} C_DIS
LIN {X 0.058,Y -187.844,Z 787.974,A 0.000,B 0.000,C 90.000,E1 355.355} C_DIS
LIN {X 0.030,Y -191.150,Z 787.942,A 0.000,B 0.000,C 90.000,E1 349.567} C_DIS
LIN {X 0.002,Y -194.565,Z 787.919,A 0.000,B 0.000,C 90.000,E1 345.463} C_DIS
LIN {X -0.058,Y -198.941,Z 787.897,A 0.000,B 0.000,C 90.000,E1 341.402} C_DIS
LIN {X -0.037,Y -204.430,Z 787.874,A 0.000,B 0.000,C 90.000,E1 337.358} C_DIS
LIN {X -0.088,Y -210.877,Z 787.852,A 0.000,B 0.000,C 90.000,E1 333.384} C_DIS
LIN {X 0.074,Y -218.226,Z 787.830,A 0.000,B 0.000,C 90.000,E1 329.410} C_DIS
LIN {X 0.050,Y -226.233,Z 787.809,A 0.000,B 0.000,C 90.000,E1 325.548} C_DIS
LIN {X 0.057,Y -234.995,Z 787.788,A 0.000,B 0.000,C 90.000,E1 321.743} C_DIS
LIN {X 0.096,Y -244.535,Z 787.767,A 0.000,B 0.000,C 90.000,E1 318.000} C_DIS
LIN {X 0.067,Y -254.937,Z 787.746,A 0.000,B 0.000,C 90.000,E1 314.352} C_DIS
LIN {X -0.024,Y -265.080,Z 787.729,A 0.000,B 0.000,C 90.000,E1 311.148} C_DIS
LIN {X 0.059,Y -276.080,Z 787.711,A 0.000,B 0.000,C 90.000,E1 307.971} C_DIS
LIN {X 0.091,Y -289.503,Z 787.692,A 0.000,B 0.000,C 90.000,E1 304.532} C_DIS
LIN {X -0.067,Y -299.868,Z 787.679,A 0.000,B 0.000,C 90.000,E1 302.212} C_DIS
LIN {X 0.201,Y -314.697,Z 787.662,A 0.000,B 0.000,C 90.000,E1 299.205} C_DIS
LIN {X 0.067,Y -329.150,Z 787.648,A 0.000,B 0.000,C 90.000,E1 296.668} C_DIS
LIN {X -0.152,Y -346.650,Z 787.633,A 0.000,B 0.000,C 90.000,E1 293.898} C_DIS
LIN {X -0.017,Y -365.895,Z 787.617,A 0.000,B 0.000,C 90.000,E1 291.153} C_DIS
LIN {X -0.088,Y -379.953,Z 787.608,A 0.000,B 0.000,C 90.000,E1 289.396} C_DIS
LIN {X -0.012,Y -399.868,Z 787.595,A 0.000,B 0.000,C 90.000,E1 287.094} C_DIS
LIN {X 0.111,Y -414.704,Z 787.586,A 0.000,B 0.000,C 90.000,E1 285.426} C_DIS
LIN {X 0.072,Y -427.035,Z 787.578,A 0.000,B 0.000,C 90.000,E1 284.064} C_DIS
LIN {X 0.111,Y -438.989,Z 787.571,A 0.000,B 0.000,C 90.000,E1 282.715} C_DIS
LIN {X 0.110,Y -448.214,Z 787.565,A 0.000,B 0.000,C 90.000,E1 281.658} C_DIS
LIN {X 0.209,Y -456.791,Z 787.559,A 0.000,B 0.000,C 90.000,E1 280.602} C_DIS
LIN {X -0.132,Y -464.786,Z 787.553,A 0.000,B 0.000,C 90.000,E1 279.613} C_DIS
LIN {X 0.075,Y -472.165,Z 787.548,A 0.000,B 0.000,C 90.000,E1 278.568} C_DIS
LIN {X -0.168,Y -478.771,Z 787.542,A 0.000,B 0.000,C 90.000,E1 277.587} C_DIS
LIN {X -0.149,Y -483.034,Z 787.538,A 0.000,B 0.000,C 90.000,E1 276.834} C_DIS
LIN {X 0.023,Y -485.480,Z 787.535,A 0.000,B 0.000,C 90.000,E1 276.315} C_DIS
LIN {X 0.044,Y -488.438,Z 787.531,A 0.000,B 0.000,C 90.000,E1 275.568} C_DIS
LIN {X -0.240,Y -490.031,Z 787.528,A 0.000,B 0.000,C 90.000,E1 275.106} C_DIS
LIN {X -0.028,Y -491.229,Z 787.525,A 0.000,B 0.000,C 90.000,E1 274.588} C_DIS
LIN {X 0.158,Y -492.017,Z 787.523,A 0.000,B 0.000,C 90.000,E1 274.073} C_DIS
LIN {X -0.106,Y -492.442,Z 787.520,A 0.000,B 0.000,C 90.000,E1 273.612} C_DIS
LIN {X 0.123,Y -492.422,Z 787.517,A 0.000,B 0.000,C 90.000,E1 273.094} C_DIS
LIN {X -0.165,Y -491.972,Z 787.515,A 0.000,B 0.000,C 90.000,E1 272.636} C_DIS
LIN {X 0.042,Y -491.134,Z 787.512,A 0.000,B 0.000,C 90.000,E1 272.121} C_DIS
LIN {X -0.226,Y -489.898,Z 787.509,A 0.000,B 0.000,C 90.000,E1 271.661} C_DIS
LIN {X -0.027,Y -488.194,Z 787.506,A 0.000,B 0.000,C 90.000,E1 271.146} C_DIS
LIN {X 0.167,Y -486.043,Z 787.504,A 0.000,B 0.000,C 90.000,E1 270.630} C_DIS
LIN {X -0.135,Y -483.314,Z 787.501,A 0.000,B 0.000,C 90.000,E1 270.172} C_DIS
LIN {X 0.029,Y -480.027,Z 787.498,A 0.000,B 0.000,C 90.000,E1 269.656} C_DIS
LIN {X 0.173,Y -475.980,Z 787.495,A 0.000,B 0.000,C 90.000,E1 269.141} C_DIS
LIN {X -0.179,Y -471.012,Z 787.493,A 0.000,B 0.000,C 90.000,E1 268.682} C_DIS
LIN {X 0.115,Y -465.084,Z 787.490,A 0.000,B 0.000,C 90.000,E1 268.165} C_DIS
LIN {X -0.183,Y -462.052,Z 787.489,A 0.000,B 0.000,C 90.000,E1 267.993} C_DIS
LIN {X -0.018,Y -458.580,Z 787.488,A 0.000,B 0.000,C 90.000,E1 267.764} C_DIS
LIN {X -0.041,Y -451.301,Z 787.486,A 0.000,B 0.000,C 90.000,E1 267.421} C_DIS
LIN {X 0.044,Y -443.722,Z 787.484,A 0.000,B 0.000,C 90.000,E1 267.135} C_DIS
LIN {X 0.201,Y -435.615,Z 787.483,A 0.000,B 0.000,C 90.000,E1 266.906} C_DIS
LIN {X 0.111,Y -431.739,Z 787.483,A 0.000,B 0.000,C 90.000,E1 266.846} C_DIS
LIN {X -0.150,Y -422.273,Z 787.482,A 0.000,B 0.000,C 90.000,E1 266.788} C_DIS
LIN {X 0.196,Y -420.224,Z 787.482,A 0.000,B 0.000,C 90.000,E1 266.731} C_DIS
LIN {X 0.052,Y -180.967,Z 787.482,A 0.000,B 0.000,C 90.000,E1 266.731} C_DIS
LIN {X 0.043,Y -180.866,Z 787.472,A 0.000,B 0.000,C 90.000,E1 265.008} C_DIS
LIN {X -0.080,Y -178.981,Z 787.444,A 0.000,B 0.000,C 90.000,E1 259.982} C_DIS
LIN {X -0.069,Y -177.952,Z 787.435,A 0.000,B 0.000,C 90.000,E1 258.285} C_DIS
LIN {X -0.049,Y -175.594,Z 787.411,A 0.000,B 0.000,C 90.000,E1 254.031} C_DIS
LIN {X -0.036,Y -172.318,Z 787.387,A 0.000,B 0.000,C 90.000,E1 249.752} C_DIS
LIN {X -0.058,Y -171.796,Z 787.383,A 0.000,B 0.000,C 90.000,E1 248.901} C_DIS
LIN {X -0.020,Y -169.468,Z 787.368,A 0.000,B 0.000,C 90.000,E1 246.305} C_DIS
LIN {X 0.035,Y -166.796,Z 787.349,A 0.000,B 0.000,C 90.000,E1 242.820} C_DIS
LIN {X 0.031,Y -162.776,Z 787.325,A 0.000,B 0.000,C 90.000,E1 238.456} C_DIS
LIN {X 0.006,Y -161.465,Z 787.315,A 0.000,B 0.000,C 90.000,E1 236.707} C_DIS
LIN {X 0.048,Y -157.460,Z 787.290,A 0.000,B 0.000,C 90.000,E1 232.271} C_DIS
LIN {X -0.020,Y -155.471,Z 787.276,A 0.000,B 0.000,C 90.000,E1 229.622} C_DIS
LIN {X 0.021,Y -151.783,Z 787.251,A 0.000,B 0.000,C 90.000,E1 225.121} C_DIS
LIN {X -0.073,Y -149.990,Z 787.236,A 0.000,B 0.000,C 90.000,E1 222.447} C_DIS
LIN {X -0.041,Y -146.822,Z 787.210,A 0.000,B 0.000,C 90.000,E1 217.890} C_DIS
LIN {X 0.065,Y -145.401,Z 787.195,A 0.000,B 0.000,C 90.000,E1 215.105} C_DIS
LIN {X -0.018,Y -142.834,Z 787.170,A 0.000,B 0.000,C 90.000,E1 210.541} C_DIS
LIN {X 0.038,Y -141.448,Z 787.149,A 0.000,B 0.000,C 90.000,E1 206.821} C_DIS
LIN {X -0.048,Y -139.370,Z 787.113,A 0.000,B 0.000,C 90.000,E1 200.355} C_DIS
LIN {X 0.069,Y -138.819,Z 787.097,A 0.000,B 0.000,C 90.000,E1 197.511} C_DIS
LIN {X -0.017,Y -138.352,Z 787.056,A 0.000,B 0.000,C 90.000,E1 190.074} C_DIS
LIN {X -0.044,Y -139.535,Z 787.004,A 0.000,B 0.000,C 90.000,E1 180.745} C_DIS
LIN {X 0.049,Y -141.221,Z 786.973,A 0.000,B 0.000,C 90.000,E1 175.122} C_DIS
LIN {X 0.008,Y -142.594,Z 786.958,A 0.000,B 0.000,C 90.000,E1 172.356} C_DIS
LIN {X -0.039,Y -144.897,Z 786.932,A 0.000,B 0.000,C 90.000,E1 167.757} C_DIS
LIN {X -0.086,Y -147.525,Z 786.911,A 0.000,B 0.000,C 90.000,E1 164.102} C_DIS
LIN {X -0.012,Y -150.121,Z 786.891,A 0.000,B 0.000,C 90.000,E1 160.423} C_DIS
LIN {X -0.001,Y -153.483,Z 786.871,A 0.000,B 0.000,C 90.000,E1 156.794} C_DIS
LIN {X 0.064,Y -157.847,Z 786.846,A 0.000,B 0.000,C 90.000,E1 152.281} C_DIS
LIN {X 0.020,Y -162.133,Z 786.826,A 0.000,B 0.000,C 90.000,E1 148.742} C_DIS
LIN {X -0.001,Y -166.337,Z 786.807,A 0.000,B 0.000,C 90.000,E1 145.229} C_DIS
LIN {X 0.005,Y -171.353,Z 786.787,A 0.000,B 0.000,C 90.000,E1 141.743} C_DIS
LIN {X -0.068,Y -176.257,Z 786.768,A 0.000,B 0.000,C 90.000,E1 138.324} C_DIS
LIN {X 0.051,Y -180.541,Z 786.754,A 0.000,B 0.000,C 90.000,E1 135.729} C_DIS
LIN {X 0.030,Y -185.943,Z 786.735,A 0.000,B 0.000,C 90.000,E1 132.366} C_DIS
LIN {X -0.035,Y -190.573,Z 786.722,A 0.000,B 0.000,C 90.000,E1 129.886} C_DIS
LIN {X -0.009,Y -192.536,Z 786.715,A 0.000,B 0.000,C 90.000,E1 128.705} C_DIS
LIN {X -0.049,Y -292.493,Z 786.715,A 0.000,B 0.000,C 90.000,E1 128.705} C_DIS
LIN {X -0.109,Y -294.834,Z 786.715,A 0.000,B 0.000,C 90.000,E1 128.669} C_DIS
LIN {X -0.143,Y -298.891,Z 786.714,A 0.000,B 0.000,C 90.000,E1 128.463} C_DIS
LIN {X 0.010,Y -301.288,Z 786.712,A 0.000,B 0.000,C 90.000,E1 128.222} C_DIS
LIN {X -0.103,Y -305.109,Z 786.709,A 0.000,B 0.000,C 90.000,E1 127.729} C_DIS
LIN {X 0.093,Y -306.814,Z 786.708,A 0.000,B 0.000,C 90.000,E1 127.363} C_DIS
LIN {X -0.141,Y -308.151,Z 786.706,A 0.000,B 0.000,C 90.000,E1 127.076} C_DIS
LIN {X -0.102,Y -319.154,Z 786.686,A 0.000,B 0.000,C 90.000,E1 123.499} C_DIS
LIN {X 0.150,Y -329.432,Z 786.670,A 0.000,B 0.000,C 90.000,E1 120.590} C_DIS
LIN {X 0.209,Y -341.051,Z 786.654,A 0.000,B 0.000,C 90.000,E1 117.769} C_DIS
LIN {X 0.127,Y -354.118,Z 786.639,A 0.000,B 0.000,C 90.000,E1 115.027} C_DIS
LIN {X 0.046,Y -367.040,Z 786.626,A 0.000,B 0.000,C 90.000,E1 112.642} C_DIS
LIN {X -0.002,Y -381.288,Z 786.613,A 0.000,B 0.000,C 90.000,E1 110.301} C_DIS
LIN {X 0.045,Y -396.966,Z 786.600,A 0.000,B 0.000,C 90.000,E1 108.000} C_DIS
LIN {X -0.142,Y -414.185,Z 786.588,A 0.000,B 0.000,C 90.000,E1 105.788} C_DIS
LIN {X -0.022,Y -433.073,Z 786.576,A 0.000,B 0.000,C 90.000,E1 103.592} C_DIS
LIN {X -0.017,Y -453.117,Z 786.564,A 0.000,B 0.000,C 90.000,E1 101.535} C_DIS
LIN {X 0.153,Y -468.403,Z 786.556,A 0.000,B 0.000,C 90.000,E1 100.084} C_DIS
LIN {X 0.133,Y -470.355,Z 786.555,A 0.000,B 0.000,C 90.000,E1 99.849} C_DIS
LIN {X 0.111,Y -471.840,Z 786.553,A 0.000,B 0.000,C 90.000,E1 99.613} C_DIS
LIN {X -0.034,Y -473.032,Z 786.552,A 0.000,B 0.000,C 90.000,E1 99.378} C_DIS
LIN {X -0.257,Y -473.901,Z 786.551,A 0.000,B 0.000,C 90.000,E1 99.151} C_DIS
LIN {X -0.068,Y -474.821,Z 786.548,A 0.000,B 0.000,C 90.000,E1 98.624} C_DIS
LIN {X 0.055,Y -474.762,Z 786.545,A 0.000,B 0.000,C 90.000,E1 98.106} C_DIS
LIN {X 0.185,Y -473.721,Z 786.542,A 0.000,B 0.000,C 90.000,E1 97.587} C_DIS
LIN {X 0.046,Y -472.785,Z 786.541,A 0.000,B 0.000,C 90.000,E1 97.352} C_DIS
LIN {X -0.153,Y -471.517,Z 786.539,A 0.000,B 0.000,C 90.000,E1 97.125} C_DIS
LIN {X -0.178,Y -452.232,Z 786.522,A 0.000,B 0.000,C 90.000,E1 94.069} C_DIS
LIN {X -0.091,Y -441.699,Z 786.512,A 0.000,B 0.000,C 90.000,E1 92.236} C_DIS
LIN {X 0.070,Y -432.491,Z 786.504,A 0.000,B 0.000,C 90.000,E1 90.630} C_DIS
LIN {X 0.180,Y -421.384,Z 786.493,A 0.000,B 0.000,C 90.000,E1 88.740} C_DIS
LIN {X 0.083,Y -410.073,Z 786.483,A 0.000,B 0.000,C 90.000,E1 86.846} C_DIS
LIN {X 0.124,Y -400.328,Z 786.473,A 0.000,B 0.000,C 90.000,E1 85.179} C_DIS
LIN {X 0.085,Y -385.727,Z 786.459,A 0.000,B 0.000,C 90.000,E1 82.648} C_DIS
LIN {X 0.170,Y -373.207,Z 786.446,A 0.000,B 0.000,C 90.000,E1 80.330} C_DIS
LIN {X -0.063,Y -355.210,Z 786.427,A 0.000,B 0.000,C 90.000,E1 76.825} C_DIS
LIN {X 0.007,Y -345.054,Z 786.415,A 0.000,B 0.000,C 90.000,E1 74.700} C_DIS
LIN {X 0.032,Y -333.633,Z 786.401,A 0.000,B 0.000,C 90.000,E1 72.236} C_DIS
LIN {X 0.151,Y -321.095,Z 786.386,A 0.000,B 0.000,C 90.000,E1 69.390} C_DIS
LIN {X 0.068,Y -306.470,Z 786.366,A 0.000,B 0.000,C 90.000,E1 65.869} C_DIS
LIN {X 0.131,Y -293.143,Z 786.346,A 0.000,B 0.000,C 90.000,E1 62.231} C_DIS
LIN {X 0.138,Y -284.153,Z 786.331,A 0.000,B 0.000,C 90.000,E1 59.537} C_DIS
LIN {X -0.004,Y -275.645,Z 786.316,A 0.000,B 0.000,C 90.000,E1 56.834} C_DIS
LIN {X -0.048,Y -267.396,Z 786.300,A 0.000,B 0.000,C 90.000,E1 54.069} C_DIS
LIN {X 0.004,Y -261.277,Z 786.289,A 0.000,B 0.000,C 90.000,E1 51.949} C_DIS
LIN {X 0.018,Y -253.160,Z 786.273,A 0.000,B 0.000,C 90.000,E1 49.094} C_DIS
LIN {X -0.070,Y -243.389,Z 786.253,A 0.000,B 0.000,C 90.000,E1 45.486} C_DIS
LIN {X -0.050,Y -235.984,Z 786.236,A 0.000,B 0.000,C 90.000,E1 42.528} C_DIS
LIN {X 0.046,Y -227.003,Z 786.215,A 0.000,B 0.000,C 90.000,E1 38.749} C_DIS
LIN {X -0.033,Y -218.518,Z 786.194,A 0.000,B 0.000,C 90.000,E1 34.945} C_DIS
LIN {X 0.106,Y -212.195,Z 786.177,A 0.000,B 0.000,C 90.000,E1 31.799} C_DIS
LIN {X -0.056,Y -206.507,Z 786.159,A 0.000,B 0.000,C 90.000,E1 28.693} C_DIS
LIN {X 0.088,Y -201.556,Z 786.142,A 0.000,B 0.000,C 90.000,E1 25.463} C_DIS
LIN {X -0.020,Y -196.385,Z 786.119,A 0.000,B 0.000,C 90.000,E1 21.461} C_DIS
LIN {X -0.083,Y -192.321,Z 786.097,A 0.000,B 0.000,C 90.000,E1 17.402} C_DIS
LIN {X 0.092,Y -188.869,Z 786.069,A 0.000,B 0.000,C 90.000,E1 12.411} C_DIS
LIN {X -0.067,Y -186.532,Z 786.028,A 0.000,B 0.000,C 90.000,E1 4.992} C_DIS
LIN {X 0.064,Y -187.997,Z 785.974,A 0.000,B 0.000,C 90.000,E1 355.355} C_DIS
LIN {X 0.007,Y -191.290,Z 785.942,A 0.000,B 0.000,C 90.000,E1 349.577} C_DIS
LIN {X 0.019,Y -194.704,Z 785.919,A 0.000,B 0.000,C 90.000,E1 345.463} C_DIS
LIN {X -0.037,Y -199.083,Z 785.897,A 0.000,B 0.000,C 90.000,E1 341.402} C_DIS
LIN {X -0.011,Y -204.595,Z 785.874,A 0.000,B 0.000,C 90.000,E1 337.358} C_DIS
LIN {X 0.034,Y -209.670,Z 785.856,A 0.000,B 0.000,C 90.000,E1 334.152} C_DIS
LIN {X 0.056,Y -216.845,Z 785.835,A 0.000,B 0.000,C 90.000,E1 330.205} C_DIS
LIN {X -0.036,Y -223.092,Z 785.817,A 0.000,B 0.000,C 90.000,E1 327.120} C_DIS
LIN {X -0.034,Y -231.506,Z 785.796,A 0.000,B 0.000,C 90.000,E1 323.290} C_DIS
LIN {X -0.089,Y -240.710,Z 785.775,A 0.000,B 0.000,C 90.000,E1 319.542} C_DIS
LIN {X 0.098,Y -250.730,Z 785.755,A 0.000,B 0.000,C 90.000,E1 315.810} C_DIS
LIN {X 0.090,Y -261.614,Z 785.735,A 0.000,B 0.000,C 90.000,E1 312.204} C_DIS
LIN {X 0.115,Y -273.523,Z 785.715,A 0.000,B 0.000,C 90.000,E1 308.669} C_DIS
